BC00472=140020,825224,1075175
BC00473=143607,831260,1075175
BC00474=145042,833675,1075175
BC00475=145042,833669,1075175
BC00476=143607,831255,1075175
BC00477=140021,825218,1075175
BC00478=140020,825224,1075175
BC00479=325300,955877,1075175
BC00480=326098,960603,1075175
BC00481=326417,962494,1075175
BC00482=373942,970744,1075175
BC00483=373623,968854,1075175
BC00484=372825,964128,1075175
BC00485=388713,844195,1075175
BC00486=388713,844195,1075175
BC00487=388713,844195,1075175
BC00488=388713,844195,1075175
BC00489=388713,844195,1075175
BC00490=392621,845560,1075175
BC00491=388844,869736,1075175
BC00492=388844,869736,1075175
BC00493=388844,869736,1075175
BC00494=388844,869736,1075175
BC00495=386515,859937,1075175
BC00496=382579,861240,1075175
BC00497=382579,861240,1075175
BC00498=398174,862085,1075175
BC00499=398174,860729,1075175
BC00500=398175,860364,1075172
BC00501=398174,860364,1075175
BC00502=398174,860364,1075175
BC00503=398174,860364,1075175
BC00504=398174,859798,1075175
BC00505=398174,853900,1075175
BC00506=335556,962122,1075175
BC00507=313093,960913,1075175
BC00508=312779,966350,1075175
BC00509=312653,968525,1075175
BC00510=317356,969341,1075175
BC00511=322596,970251,1075175
BC00512=322722,968076,1075175
BC00513=323035,962639,1075175
BC00514=275790,965253,1075175
BC00515=219096,968390,1075175
BC00516=223120,970377,1075175
BC00517=224729,971172,1075175
BC00518=220819,966503,1075175
BC00519=219210,965708,1075175
BC00520=215186,963721,1075175
BC00521=283252,975030,1075175
BC00522=343583,985054,1075175
BC00523=351318,986339,1075175
BC00524=346951,987672,1075175
BC00525=345577,987893,1075175
BC00526=346840,986833,1075175
BC00527=348087,985787,1075175
BC00528=349722,984415,1075175
BC00529=349722,984415,1075175
BC00530=349722,984415,1075175
BC00531=351469,983882,1075175
BC00532=355836,982549,1075175
BC00533=351318,986339,1075175
BC00534=322594,894090,1075175
BC00535=319270,885244,1075175
BC00536=319145,881395,1075175
BC00537=319096,879856,1075175
BC00538=319096,879856,1075175
BC00539=310158,881364,1075175
BC00540=310282,885213,1075175
BC00541=287932,898047,1075175
BC00542=289217,893542,1075175
BC00543=289730,891739,1075175
BC00544=285692,891718,1075175
BC00545=285179,893520,1075175
BC00546=283894,898026,1075175
BC00547=317886,904348,1075175
BC00548=321408,904356,1075175
BC00549=251917,914686,1075175
BC00550=191223,885215,1075175
BC00551=191223,923708,1075175
BC00552=186619,926680,1075175
BC00553=184777,927869,1075175
BC00554=132357,904545,1075175
BC00555=148459,907340,1075175
BC00556=150318,907039,1075175
BC00557=172119,903510,1075175
BC00558=172334,901853,1075175
BC00559=172871,897709,1075175
BC00560=285135,920733,1075175
BC00561=282294,924718,1075175
BC00562=278369,925274,1075175
BC00563=250842,915028,1075175
BC00564=302481,924098,1075175
BC00565=235391,926007,1075175
BC00566=233206,924435,1075175
BC00567=227742,920504,1075175
BC00568=172871,874776,1075175
BC00569=140749,823212,1075175
BC00570=114392,780903,1075175
BC00571=114392,780903,1075175
BC00572=114392,780903,1075175
BC00573=114392,780903,1075175
BC00574=114392,780903,1075175
BC00575=114392,780903,1075175
BC00576=114392,780903,1075175
BC00577=114392,780903,1075175
BC00578=147421,791636,1075175
BC00579=157474,794903,1075175
BC00580=157474,794903,1075175
BC00581=157474,794903,1075175
BC00582=157474,794903,1075175
BC00583=157474,794903,1075175
BC00584=157474,794903,1075175
BC00585=157474,794903,1075175
BC00586=157474,794903,1075175
BC00587=188976,808930,1075175
BC00588=188976,808930,1075175
BC00589=188976,808930,1075175
BC00590=188976,808930,1075175
BC00591=188976,808930,1075175
BC00592=188976,808930,1075175
BC00593=188976,808930,1075175
BC00594=188976,808930,1075175
BC00595=147641,782026,1075175
BC00596=198576,845167,1075175
BC00597=232811,933878,1075175
BC00598=232896,933343,1075175
BC00599=232035,938717,1075175
BC00600=231691,940867,1075175
BC00601=233684,941999,1075172
BC00602=218918,951560,1075175
BC00603=218487,945823,1075175
BC00604=199715,965567,1075175
BC00605=202231,971242,1075175
BC00606=203237,973512,1075175
BC00607=199770,971953,1075175
BC00608=198686,969649,1075175
BC00609=195975,963887,1075175
BC00610=268319,958805,1075175
BC00611=299772,956595,1075175
BC00612=294961,960779,1075175
BC00613=302025,967105,1075175
BC00614=302025,967105,1075175
BC00615=302862,967571,1075175
BC00616=304981,965989,1075175
BC00617=310277,962032,1075175
BC00618=299772,946803,1075175
BC00619=156368,867370,1075175
BC00620=114190,943890,1075175
BC00621=112857,947238,1075175
BC00622=112324,948578,1075175
BC00623=57438,939049,1075175
BC00624=57438,939049,1075175
BC00625=57972,937710,1075175
BC00626=59304,934362,1075175
BC00627=59959,931573,1075175
BC00628=60163,930702,1075175
BC00629=64900,934429,1075175
BC00630=66794,935919,1075175
BC00631=70926,933782,1075175
BC00632=86714,920781,1075175
BC00633=88876,916896,1075175
BC00634=87247,915034,1075175
BC00635=83174,910378,1075175
BC00636=93083,910762,1075175
BC00637=96362,916987,1075175
BC00638=97673,919477,1075175
BC00639=102107,915596,1075175
BC00640=93734,925368,1075175
BC00641=92128,923198,1075175
BC00642=88115,917772,1075175
BC00643=59304,853852,1075175
BC00644=302197,956351,1075175
BC00645=302197,956351,1075175
BC00646=297684,958955,1075175
BC00647=295879,959997,1075175
BC00648=304739,998959,1075175
BC00649=304723,978619,1075175
BC00650=293949,1042099,1075175
BC00651=295296,1044279,1075175
BC00652=298665,1049727,1075175
BC00653=298665,1049727,1075175
BC00654=21214,672831,1075175
BC00655=78393,670967,1075175
BC00656=177059,727519,1002542
BC00657=78393,913126,1075175
BC00658=70793,903989,1075175
BC00659=70793,903989,1075175
BC00660=70793,903989,1075175
BC00661=70793,903989,1075175
BC00662=70793,903989,1075175
BC00663=70793,903989,1075175
BC00664=70793,903989,1075175
BC00665=70793,903989,1075175
BC00666=70793,903989,1075175
BC00667=103901,897249,1075175
BC00668=103901,897249,1075175
BC00669=103901,897249,1075175
BC00670=103901,897249,1075175
BC00671=103901,897249,1075175
BC00672=103901,897249,1075175
BC00673=103901,897249,1075175
BC00674=103901,897249,1075175
BC00675=89915,910531,1075175
BC00676=89915,910531,1075175
BC00677=89916,910530,1075174
BC00678=89916,910530,1075174
BC00679=89916,910530,1075174
BC00680=89916,910530,1075174
BC00681=89916,910530,1075174
BC00682=89916,910530,1075174
BC00683=89916,910530,1075174
BC00684=89915,910531,1075175
BC00685=89915,910531,1075175
BC00686=89915,910531,1075175
BC00687=89915,910531,1075175
BC00688=89915,910531,1075175
BC00689=89915,910531,1075175
BC00690=89915,910531,1075175
BC00691=27368,899646,1075175
BC00692=27368,899646,1075175
BC00693=27368,899646,1075175
BC00694=27368,899646,1075175
BC00695=27368,899646,1075175
BC00696=27368,899646,1075175
BC00697=27368,899646,1075175
BC00698=27368,899646,1075175
BC00699=160753,772187,1075175
BC00700=160753,772187,1075175
BC00701=160753,772187,1075175
BC00702=160753,772187,1075175
BC00703=160753,772187,1075175
BC00704=160753,772187,1075175
BC00705=160753,772187,1075175
BC00706=160753,772187,1075175
BC00707=160753,772187,1075175
BC00708=160753,772187,1075175
BC00709=160753,772187,1075175
BC00710=160753,772187,1075175
BC00711=123402,765716,1075175
BC00712=123402,765716,1075175
BC00713=123402,765716,1075175
BC00714=123402,765716,1075175
BC00715=123402,765716,1075175
BC00716=123402,765716,1075175
BC00717=123402,765716,1075175
BC00718=123402,765716,1075175
BC00719=123402,765716,1075175
BC00720=123402,765716,1075175
BC00721=123402,765716,1075175
BC00722=129464,768278,1075175
BC00723=151149,777443,1075175
BC00724=169689,785624,1075175
BC00725=169689,785624,1075175
BC00726=169689,785624,1075175
BC00727=169689,785624,1075175
BC00728=169689,785624,1075175
BC00729=169689,785624,1075175
BC00730=169689,785624,1075175
BC00731=169689,785624,1075175
BC00732=169689,785624,1075175
BC00733=169689,785624,1075175
BC00734=169689,785624,1075175
BC00735=169689,785624,1075175
BC00736=169689,785624,1075175
BC00737=120114,813651,1075175
BC00738=120114,813651,1075175
BC00739=120114,813651,1075175
BC00740=120114,813651,1075175
BC00741=120114,813651,1075175
BC00742=120114,813651,1075175
BC00743=120114,813651,1075175
BC00744=120114,813651,1075175
BC00745=120114,813651,1075175
BC00746=120114,813651,1075175
BC00747=120114,813651,1075175
BC00748=120114,813651,1075175
BC00749=120114,813651,1075175
BC00750=141881,838168,1075175
BC00751=141881,838168,1075175
BC00752=141881,838168,1075175
BC00753=141881,838168,1075175
BC00754=141881,838168,1075175
BC00755=141881,838168,1075175
BC00756=141881,838168,1075175
BC00757=141881,838168,1075175
BC00758=141881,838168,1075175
BC00759=141881,838168,1075175
BC00760=141881,838168,1075175
BC00761=141881,838168,1075175
BC00762=141881,838168,1075175
BC00763=69874,805894,1075175
BC00764=70019,750208,1075175
BC00765=70019,750208,1075175
BC00766=70019,750208,1075175
BC00767=70019,750208,1075175
BC00768=70019,750208,1075175
BC00769=70019,750208,1075175
BC00770=70019,750208,1075175
BC00771=70019,750208,1075175
BC00772=70019,750208,1075175
BC00773=70019,750208,1075175
BC00774=70019,750208,1075175
BC00775=70019,750208,1075175
BC00776=70019,750208,1075175
BC00777=70018,750208,1075172
BC00778=70018,750208,1075172
BC00779=70018,750208,1075172
BC00780=70018,750208,1075172
BC00781=70018,750208,1075172
BC00782=70018,750208,1075172
BC00783=70018,750208,1075172
BC00784=70018,750208,1075172
BC00785=110204,822960,1075174
BC00786=128430,855958,1075175
BC00787=125005,945340,1075175
BC00788=125005,945340,1075175
BC00789=125005,945340,1075175
BC00790=125005,945340,1075175
BC00791=125005,945340,1075175
BC00792=125005,945340,1075175
BC00793=125005,945340,1075175
BC00794=125005,945340,1075175
BC00795=125005,945340,1075175
BC00796=125005,945340,1075175
BC00797=125005,945340,1075175
BC00798=177748,940008,1075175
BC00799=177748,940008,1075175
BC00800=177748,940008,1075175
BC00801=177748,940008,1075175
BC00802=177748,940008,1075175
BC00803=177748,940008,1075175
BC00804=177748,940008,1075175
BC00805=177748,940008,1075175
BC00806=177748,940008,1075175
BC00807=177748,940008,1075175
BC00808=177748,940008,1075175
BC00809=177748,940008,1075175
BC00810=225975,953000,1075175
BC00811=225975,953000,1075175
BC00812=225975,953000,1075175
BC00813=225975,953000,1075175
BC00814=225975,953000,1075175
BC00815=225975,953000,1075175
BC00816=225975,953000,1075175
BC00817=225975,953000,1075175
BC00818=225975,953000,1075175
BC00819=225975,953000,1075175
BC00820=225975,953000,1075175
BC00821=225975,953000,1075175
BC00822=254413,953027,1075175
BC00823=252547,954523,1075175
BC00824=252548,954519,1075175
BC00825=252583,954651,1075175
BC00826=252019,957675,1075175
BC00827=252583,954651,1075175
BC00828=252165,954787,1075175
BC00829=249030,954243,1075175
BC00830=252165,954787,1075175
BC00831=258696,949550,1075175
BC00832=257059,950024,1075175
BC00833=265795,953000,1075175
BC00834=265795,953000,1075175
BC00835=265795,953000,1075175
BC00836=265795,953000,1075175
BC00837=265795,953000,1075175
BC00838=265795,953000,1075175
BC00839=265795,953000,1075175
BC00840=265795,953000,1075175
BC00841=265795,953000,1075175
BC00842=265795,953000,1075175
BC00843=265795,953000,1075175
BC00844=254634,951648,1075175
BC00845=253737,956448,1075175
BC00846=253378,958368,1075175
BC00847=253379,958364,1075175
BC00848=253259,958395,1075175
BC00849=252695,961419,1075175
BC00850=253259,958395,1075175
BC00851=254515,951675,1075175
BC00852=248439,993035,1075175
BC00853=271638,1017285,1075175
BC00854=314947,1062557,1075175
BC00855=311280,1056373,1075175
BC00856=310409,1054905,1075175
BC00857=310409,1054901,1075175
BC00858=310409,1054905,1075175
BC00859=284329,1066137,1075175
BC00860=285931,1063482,1075175
BC00861=284329,1066137,1075175
BC00862=333588,1039325,1075175
BC00863=330835,1037779,1075175
BC00864=333588,1039325,1075175
BC00865=340460,1045393,1075175
BC00866=319968,1046454,1075175
BC00867=279319,1048558,1075175
BC00868=281895,1044284,1075175
BC00869=282926,1042574,1075175
BC00870=282926,1042570,1075175
BC00871=282744,1042486,1075175
BC00872=284346,1039831,1075175
BC00873=282744,1042486,1075175
BC00874=279137,1048470,1075175
BC00875=253507,1028204,1074244
BC00876=253507,1028204,1074244
BC00877=253507,1028204,1074244
BC00878=253507,1028204,1074244
BC00879=253507,1028204,1074244
BC00880=253507,1028204,1074244
BC00881=253507,1028204,1074244
BC00882=253507,1028204,1074244
BC00883=253507,1028204,1074244
BC00884=253507,1028204,1074244
BC00885=253507,1028204,1074244
BC00886=253507,1028204,1074244
BC00887=253507,1028204,1074244
BC00888=212842,1022781,1075175
BC00889=146334,1015862,1075175
BC00890=66205,1045023,1075175
BC00891=66205,1045023,1075175
BC00892=66205,1045023,1075175
BC00893=66205,1045023,1075175
BC00894=66205,1045023,1075175
BC00895=66205,1045023,1075175
BC00896=66205,1045023,1075175
BC00897=66205,1045023,1075175
BC00898=66205,1045023,1075175
BC00899=66205,1045023,1075175
BC00900=66205,1045023,1075175
BC00901=66205,1045023,1075175
BC00902=125029,959783,1075175
BC00903=190390,972133,1075175
BC00904=190390,972133,1075175
BC00905=190390,972133,1075173
BC00906=190390,972133,1075175
BC00907=190390,972133,1075175
BC00908=190390,972133,1075175
BC00909=190390,972133,1075175
BC00910=190390,972133,1075175
BC00911=190390,972133,1075175
BC00912=190390,972133,1075175
BC00913=190390,972133,1075175
BC00914=190390,972133,1075175
BC00915=190390,972133,1075175
BC00916=103363,888035,1075175
BC00917=35304,822265,1075175
BC00918=35304,822265,1075175
BC00919=35304,822265,1075175
BC00920=35304,822265,1075175
BC00921=35304,822265,1075175
BC00922=35304,822265,1075175
BC00923=35304,822265,1075175
BC00924=35304,822265,1075175
BC00925=35304,822265,1075175
BC00926=35304,822265,1075175
BC00927=35304,822265,1075175
BC00928=35304,822265,1075175
BC00929=167967,799945,1075175
BC00930=311305,898961,1075175
BC00931=311305,898961,1075175
BC00932=311305,898961,1075175
BC00933=311305,898961,1075175
BC00934=311305,898961,1075175
BC00935=311305,898961,1075175
BC00936=311305,898961,1075175
BC00937=311305,898961,1075175
BC00938=311305,898961,1075175
BC00939=311305,898961,1075175
BC00940=311305,898961,1075175
BC00941=311305,898961,1075175
BC00942=113180,824290,1075229
BC00943=113180,824290,1075229
BC00944=113180,824290,1075229
BC00945=113180,824290,1075229
BC00946=113180,824290,1075229
BC00947=113180,824290,1075229
BC00948=113180,824290,1075229
BC00949=113180,824290,1075229
BC00950=113180,824290,1075229
BC00951=113180,824290,1075229
BC00952=113180,824290,1075229
BC00953=113180,824290,1075229
BC00954=355762,967535,1075175
BC00955=355762,967535,1075175
BC00956=355762,967535,1075175
BC00957=355762,967535,1075175
BC00958=355762,967535,1075175
BC00959=355762,967535,1075175
BC00960=355762,967535,1075175
BC00961=355762,967535,1075175
BC00962=397203,974799,1075175
BC00963=397203,974799,1075175
BC00964=397203,974799,1075175
BC00965=397203,974799,1075175
BC00966=397203,974799,1075175
BC00967=397203,974799,1075175
BC00968=397203,974799,1075175
BC00969=397203,974799,1075175
BC00970=389868,1004990,1075175
BC00971=389868,1004990,1075175
BC00972=389868,1004990,1075175
BC00973=389868,1004990,1075175
BC00974=389868,1004990,1075175
BC00975=389868,1004990,1075175
BC00976=397203,974799,1075175
BC00977=279782,952911,1075175
BC00978=264332,967435,1075175
BC00979=264332,967435,1075175
BC00980=264332,967435,1075175
BC00981=264332,967435,1075175
BC00982=264332,967435,1075175
BC00983=264332,967435,1075175
BC00984=264332,967435,1075175
BC00985=264332,967435,1075175
BC00986=264332,967435,1075175
BC00987=264332,967435,1075175
BC00988=264332,967435,1075175
BC00989=290594,956201,1075175
BC00990=316856,944967,1075175
BC00991=316856,944967,1075175
BC00992=316856,944967,1075175
BC00993=316856,944967,1075175
BC00994=316856,944967,1075175
BC00995=316856,944967,1075175
BC00996=316856,944967,1075175
BC00997=316856,944967,1075175
BC00998=316856,944967,1075175
BC00999=316856,944967,1075175
BC01000=316856,944967,1075175
BC01001=316856,944967,1075175
BC01002=316856,944967,1075175
BC01003=316856,944967,1075175
BC01004=316856,944967,1075175
BC01005=316856,944967,1075175
BC01006=329946,891084,1075175
BC01007=337525,859888,1075175
BC01008=337525,859888,1075175
BC01009=337525,859888,1075175
BC01010=337525,859888,1075175
BC01011=337525,859888,1075175
BC01012=337525,859888,1075175
BC01013=337525,859888,1075175
BC01014=337525,859888,1075175
BC01015=238148,874377,1075175
BC01016=227206,875826,1075175
BC01017=227206,875826,1075175
BC01018=227206,875826,1075175
BC01019=227206,875826,1075175
BC01020=227206,875826,1075175
BC01021=227206,875826,1075175
BC01022=280946,887675,1075175
BC01023=280946,887675,1075175
BC01024=280946,887675,1075175
BC01025=280946,887675,1075175
BC01026=280946,887675,1075175
BC01027=280946,887675,1075175
BC01028=280946,887675,1075175
BC01029=280946,887675,1075175
BC01030=239261,850045,1075175
BC01031=207869,857354,1075175
BC01032=207869,857354,1075175
BC01033=207869,857354,1075175
BC01034=207869,857354,1075175
BC01035=207869,857354,1075175
BC01036=207869,857354,1075175
BC01037=207869,857354,1075175
BC01038=207869,857354,1075175
BC01039=207996,857850,1075175
BC01040=184532,936508,1075175
BC01041=203495,1021788,1075175
BC01042=203934,1024782,1075175
BC01043=204108,1022909,1075171
BC01044=204109,1022908,1075172
BC01045=193998,1019034,1075175
BC01046=193559,1023720,1075175
BC01047=122539,997675,1075175
BC01048=122539,997675,1075175
BC01049=122540,997675,1075169
BC01050=122540,997675,1075169
BC01051=122539,997675,1075175
BC01052=122539,997675,1075175
BC01053=110261,971952,1075175
BC01054=110261,971952,1075175
BC01055=110261,971952,1075175
BC01056=110261,971952,1075175
BC01057=110261,971952,1075175
BC01058=110261,971952,1075175
BC01059=222038,980891,1075175
BC01060=314817,1023461,1075175
BC01061=333143,1031869,1075175
BC01062=333143,1031869,1075175
BC01063=333143,1031869,1075175
BC01064=333143,1031869,1075175
BC01065=333143,1031869,1075175
BC01066=163675,1006427,1075175
BC01067=163675,1006427,1075175
BC01068=164114,1001741,1075175
BC01069=164289,999867,1075175
BC01070=160191,997498,1075175
BC01071=158450,996490,1075175
BC01072=154353,994119,1075175
BC01073=154178,995993,1075175
BC01074=153739,1000679,1075175
BC01075=82719,974634,1075175
BC01076=82719,974634,1075175
BC01077=82720,974634,1075172
BC01078=82720,974634,1075172
BC01079=82719,974634,1075175
BC01080=82720,974634,1075173
BC01081=82719,974634,1075175
BC01082=82719,974634,1075175
BC01083=70441,948911,1075175
BC01084=70441,948911,1075175
BC01085=70441,948911,1075175
BC01086=70441,948911,1075175
BC01087=70441,948911,1075175
BC01088=70441,948911,1075175
BC01089=182218,957850,1075175
BC01090=274997,1000420,1075175
BC01091=293323,1008828,1075175
BC01092=293323,1008828,1075175
BC01093=293323,1008828,1075175
BC01094=293323,1008828,1075175
BC01095=293323,1008828,1075175
BC01096=293323,1008828,1075175
BC01097=337244,1059629,1075175
BC01098=337244,1059629,1075175
BC01099=337244,1059629,1075175
BC01100=337244,1059629,1075175
BC01101=337244,1059629,1075175
BC01102=337244,1059629,1075175
BC01103=337244,1059629,1075175
BC01104=227430,982125,1075175
BC01105=115014,939685,1075175
BC01106=118867,937244,1075175
BC01107=120408,936268,1075175
BC01108=140995,947826,1075175
BC01109=182041,976368,1075175
BC01110=180846,977671,1075175
BC01111=177859,980929,1075175
BC01112=194800,984537,1075175
BC01113=244653,1016084,1075175
BC01114=241511,1010564,1075175
BC01115=240254,1008357,1075175
BC01116=240254,1008354,1075175
BC01117=241511,1010562,1075175
BC01118=244653,1016081,1075175
BC01119=244653,1016084,1075175
BC01120=272695,1033702,1075175
BC01121=285514,1041756,1075175
BC01122=284751,1045931,1075175
BC01123=282162,1039999,1075175
BC01124=281126,1037626,1075175
BC01125=207140,1028015,1075175
BC01126=213441,1031536,1075175
BC01127=213388,1030834,1075175
BC01128=213388,1030834,1075175
BC01129=212628,1031081,1075217
BC01130=212628,1031081,1075217
BC01131=212628,1031081,1075217
BC01132=212628,1031081,1075217
BC01133=212628,1031081,1075202
BC01134=202210,1012854,1075175
BC01135=202210,1012854,1075175
BC01136=196613,982513,1075175
BC01137=175963,870568,1075175
BC01138=163612,803610,1075175
BC01139=152631,778532,1075175
BC01140=146092,780306,1075175
BC01141=143477,781016,1075175
BC01142=143597,781078,1075175
BC01143=143625,781092,1075175
BC01144=143746,781156,1075175
BC01145=146361,780446,1075175
BC01146=152900,778672,1075175
BC01147=152900,778672,1075175
BC01148=74084,744686,1075175
BC01149=74084,744686,1075175
BC01150=67287,679894,1075175
BC01151=67287,679894,1075175
BC01152=67287,679894,1075175
BC01153=67287,679894,1075175
BC01154=67287,679894,1075175
BC01155=67287,679894,1075175
BC01156=67287,679894,1075175
BC01157=67287,679894,1075175
BC01158=83395,694294,1075175
BC01159=102108,711022,1075175
BC01160=165558,767742,1075175
BC01161=222482,818628,1075175
BC01162=215814,820321,1075175
BC01163=213147,820999,1075175
BC01164=213147,820994,1075175
BC01165=213147,820993,1075175
BC01166=213148,820988,1075175
BC01167=215815,820311,1075175
BC01168=222483,818617,1075175
BC01169=173722,816110,1075175
BC01170=90356,811823,1075175
BC01171=89696,811574,1075175
BC01172=89432,811475,1075175
BC01173=89432,811475,1075175
BC01174=89432,811475,1075175
BC01175=85301,809160,1075175
BC01176=73323,802435,1075175
BC01177=69196,800114,1075175
BC01178=69460,800213,1075175
BC01179=70120,800462,1075175
BC01180=203969,867991,1075175
BC01181=200192,866637,1075175
BC01182=198681,866095,1075175
BC01183=196278,870078,1075175
BC01184=188025,883752,1075175
BC01185=185620,887734,1075175
BC01186=187131,888276,1075175
BC01187=190907,889630,1075175
BC01188=185807,834457,1075175
BC01189=185042,826181,1075175
BC01190=182820,831186,1075175
BC01191=181931,833188,1075175
BC01192=205283,846231,1075175
BC01193=246906,863634,1075175
BC01194=246906,863634,1075175
BC01195=248214,861732,1075175
BC01196=251484,856977,1075175
BC01197=177002,833071,1075175
BC01198=153563,828435,1075175
BC01199=140020,825224,1075175
BC01200=143607,831260,1075175
BC01201=145042,833675,1075175
BC01202=145042,833669,1075175
BC01203=143607,831255,1075175
BC01204=140021,825218,1075175
BC01205=140020,825224,1075175
BC01206=325300,955877,1075175
BC01207=326098,960603,1075175
BC01208=326417,962494,1075175
BC01209=373942,970744,1075175
BC01210=373934,970699,1075175
BC01211=373927,970659,1075175
BC01212=372825,964128,1075175
BC01213=388713,844195,1075175
BC01214=388713,844195,1075175
BC01215=388713,844195,1075175
BC01216=388713,844195,1075175
BC01217=388713,844195,1075175
BC01218=392621,845560,1075175
BC01219=388844,869736,1075175
BC01220=388844,869736,1075175
BC01221=388844,869736,1075175
BC01222=388844,869736,1075175
BC01223=386515,859937,1075175
BC01224=382579,861240,1075175
BC01225=382579,861240,1075175
BC01226=398174,862085,1075175
BC01227=398174,860729,1075175
BC01228=398175,860364,1075172
BC01229=398174,860364,1075175
BC01230=398174,860364,1075175
BC01231=398174,860364,1075175
BC01232=398174,859798,1075175
BC01233=398174,853900,1075175
BC01234=335556,962122,1075175
BC01235=313093,960913,1075175
BC01236=312779,966350,1075175
BC01237=312653,968525,1075175
BC01238=317356,969341,1075175
BC01239=322596,970251,1075175
BC01240=322722,968076,1075175
BC01241=323035,962639,1075175
BC01242=275790,965253,1075175
BC01243=219096,968390,1075175
BC01244=223120,970377,1075175
BC01245=224729,971172,1075175
BC01246=220819,966503,1075175
BC01247=219210,965708,1075175
BC01248=215186,963721,1075175
BC01249=283252,975030,1075175
BC01250=343583,985054,1075175
BC01251=351318,986339,1075175
BC01252=346951,987672,1075175
BC01253=345577,987893,1075175
BC01254=346840,986833,1075175
BC01255=348087,985787,1075175
BC01256=349722,984415,1075175
BC01257=349722,984415,1075175
BC01258=349722,984415,1075175
BC01259=351469,983882,1075175
BC01260=355836,982549,1075175
BC01261=351318,986339,1075175
BC01262=375376,962122,1075175
BC01263=352913,960913,1075175
BC01264=352599,966350,1075175
BC01265=352473,968525,1075175
BC01266=357176,969341,1075175
BC01267=362416,970251,1075175
BC01268=362542,968076,1075175
BC01269=362855,962639,1075175
BC01270=315610,965253,1075175
BC01271=258916,968390,1075175
BC01272=262940,970377,1075175
BC01273=264549,971172,1075175
BC01274=260639,966503,1075175
BC01275=259030,965708,1075175
BC01276=255006,963721,1075175
BC01277=323072,975030,1075175
BC01278=383403,985054,1075175
BC01279=391138,986339,1075175
BC01280=386771,987672,1075175
BC01281=385397,987893,1075175
BC01282=386660,986833,1075175
BC01283=387907,985787,1075175
BC01284=389542,984415,1075175
BC01285=389542,984415,1075175
BC01286=389542,984415,1075175
BC01287=391289,983882,1075175
BC01288=394785,983280,1075175
BC01289=393350,984484,1075175
BC01290=322594,894090,1075175
BC01291=319270,885244,1075175
BC01292=319145,881395,1075175
BC01293=319096,879856,1075175
BC01294=319096,879856,1075175
BC01295=310158,881364,1075175
BC01296=310282,885213,1075175
BC01297=287932,898047,1075175
BC01298=289217,893542,1075175
BC01299=289730,891739,1075175
BC01300=285692,891718,1075175
BC01301=285179,893520,1075175
BC01302=283894,898026,1075175
BC01303=317886,904348,1075175
BC01304=321408,904356,1075175
BC01305=251917,914686,1075175
BC01306=191223,885215,1075175
BC01307=191223,923708,1075175
BC01308=186619,926680,1075175
BC01309=184777,927869,1075175
BC01310=132357,904545,1075175
BC01311=148459,907340,1075175
BC01312=150318,907039,1075175
BC01313=172119,903510,1075175
BC01314=172334,901853,1075175
BC01315=172871,897709,1075175
BC01316=285135,920733,1075175
BC01317=282294,924718,1075175
BC01318=278369,925274,1075175
BC01319=250842,915028,1075175
BC01320=259644,916574,1075175
BC01321=259644,916574,1075174
BC01322=259644,916574,1075175
BC01323=285135,920733,1075175
BC01324=320470,920733,1075175
BC01325=320470,920733,1075175
BC01326=320470,920733,1075172
BC01327=320470,920733,1075172
BC01328=320470,920733,1075172
BC01329=302481,924098,1075175
BC01330=235391,926007,1075175
BC01331=235391,926007,1075175
BC01332=227742,920504,1075175
BC01333=172871,874776,1075175
BC01334=140749,823212,1075175
BC01335=114392,780903,1075175
BC01336=114392,780903,1075175
BC01337=114392,780903,1075175
BC01338=114392,780903,1075175
BC01339=114392,780903,1075175
BC01340=114392,780903,1075175
BC01341=114392,780903,1075175
BC01342=114392,780903,1075175
BC01343=147421,791636,1075175
BC01344=157474,794903,1075175
BC01345=157474,794903,1075175
BC01346=157474,794903,1075175
BC01347=157474,794903,1075175
BC01348=157474,794903,1075175
BC01349=157474,794903,1075175
BC01350=157474,794903,1075175
BC01351=157474,794903,1075175
BC01352=188976,808930,1075175
BC01353=188976,808930,1075175
BC01354=188976,808930,1075175
BC01355=188976,808930,1075175
BC01356=188976,808930,1075175
BC01357=188976,808930,1075175
BC01358=188976,808930,1075175
BC01359=188976,808930,1075175
BC01360=147641,782026,1075175
BC01361=198576,845167,1075175
BC01362=232811,933878,1075175
BC01363=232896,933343,1075175
BC01364=232035,938717,1075175
BC01365=231691,940867,1075175
BC01366=233684,941999,1075172
BC01367=218918,951560,1075175
BC01368=218487,945823,1075175
BC01369=199715,965567,1075175
BC01370=202231,971242,1075175
BC01371=203237,973512,1075175
BC01372=199770,971953,1075175
BC01373=198686,969649,1075175
BC01374=195975,963887,1075175
BC01375=268319,958805,1075175
BC01376=299772,956595,1075175
BC01377=294961,960779,1075175
BC01378=302025,967105,1075175
BC01379=302025,967105,1075175
BC01380=302862,967571,1075175
BC01381=304981,965989,1075175
BC01382=310277,962032,1075175
BC01383=299772,946803,1075175
BC01384=156368,867370,1075175
BC01385=114190,943890,1075175
BC01386=112857,947238,1075175
BC01387=112324,948578,1075175
BC01388=112324,948578,1075175
BC01389=91893,945031,1075175
BC01390=58795,939285,1075175
BC01391=57438,939049,1075175
BC01392=57972,937710,1075175
BC01393=59304,934362,1075175
BC01394=59959,931573,1075175
BC01395=60163,930702,1075175
BC01396=64900,934429,1075175
BC01397=66794,935919,1075175
BC01398=70926,933782,1075175
BC01399=86714,920781,1075175
BC01400=88876,916896,1075175
BC01401=87247,915034,1075175
BC01402=83174,910378,1075175
BC01403=93083,910762,1075175
BC01404=96362,916987,1075175
BC01405=97673,919477,1075175
BC01406=102107,915596,1075175
BC01407=93734,925368,1075175
BC01408=92128,923198,1075175
BC01409=88115,917772,1075175
BC01410=59304,853852,1075175
BC01411=302197,956351,1075175
BC01412=302197,956351,1075175
BC01413=297684,958955,1075175
BC01414=295879,959997,1075175
BC01415=304739,998959,1075175
BC01416=304723,978619,1075175
BC01417=293949,1042099,1075175
BC01418=295296,1044279,1075175
BC01419=298665,1049727,1075175
BC01420=298665,1049727,1075175
BC01421=302197,956351,1075175
BC01422=339931,956351,1075175
BC01423=339931,956351,1075175
BC01424=339931,956351,1075175
BC01425=345108,996833,1075175
BC01426=329498,1037164,1075167
BC01427=329498,1037164,1075167
BC01428=329498,1037164,1075167
BC01429=326051,1024211,1075168
BC01430=315665,949153,1075168
BC01431=252444,896504,1075168
BC01432=116643,896504,1075168
BC01433=116643,972299,1075168
BC01434=116644,972299,1070754
BC01435=116644,972299,1070754
BC01436=121804,1001122,1070754
BC01437=121804,1001122,1070754
BC01438=121804,1001122,1070754
BC01439=121804,1001122,1070754
BC01440=164206,909682,1070754
BC01441=118737,834368,1072160
BC01442=21214,672831,1075175
BC01443=21214,672831,272422
BC01444=236199,677421,175874
BC01445=277013,737492,108841
BC01446=313151,790681,49489
BC01447=313151,790681,49489
BC01448=313151,790681,49489
BC01449=313151,790681,49489
BC01450=313151,790681,49489
BC01451=313151,790681,49489
BC01452=313151,790681,49489
BC01453=313151,790681,49489
BC01454=313151,790681,49489
BC01455=313151,790681,49489
BC01456=313151,790681,49489
BC01457=313151,790681,49489
BC01458=313151,790681,49489
BC01459=339082,790681,219047
BC01460=339082,790681,219047
BC01461=339082,790681,219047
BC01462=339082,790681,219047
BC01463=339082,790681,219047
BC01464=339082,790681,219047
BC01465=339082,790681,219047
BC01466=339082,790681,219047
BC01467=339082,790681,219047
BC01468=318756,790681,206942
BC01469=318756,790681,206942
BC01470=318756,790681,206942
BC01471=318756,790681,206942
BC01472=318756,790681,206942
BC01473=318756,790681,206942
BC01474=318756,790681,206941
BC01475=318756,790681,206941
BC01476=318756,790681,206942
BC01477=330178,790681,186109
BC01478=360333,790681,131110
BC01479=360333,790681,131110
BC01480=360333,790681,131110
BC01481=360333,790681,131110
BC01482=360333,790681,131110
BC01483=360333,790681,131110
BC01484=360333,790681,131110
BC01485=360333,790681,131110
BC01486=360333,790681,131110
BC01487=319787,790681,204440
BC01488=319787,790681,204440
BC01489=319787,790681,204440
BC01490=319787,790681,204440
BC01491=319787,790681,204440
BC01492=319787,790681,204440
BC01493=319787,790681,204440
BC01494=319787,790681,204440
BC01495=319787,790681,204440
BC01496=319787,790681,204440
BC01497=319787,790681,204440
BC01498=319787,790681,204440
BC01499=319787,790681,204440
BC01500=319787,790681,204440
BC01501=319787,790681,204440
BC01502=319787,790681,204440
BC01503=345989,790681,139065
BC01504=345989,790681,139065
BC01505=345988,790681,139065
BC01506=345988,790681,139065
BC01507=345988,790681,139065
BC01508=345988,790681,139065
BC01509=345988,790681,139065
BC01510=345988,790681,139065
BC01511=345988,790681,139065
BC01512=345988,790681,139065
BC01513=345988,790681,139065
BC01514=345988,790681,139065
BC01515=345988,790681,139065
BC01516=345988,790681,139065
BC01517=345988,790681,139065
BC01518=345989,790681,139065
BC01519=308625,748445,196549
BC01520=237635,668196,305769
BC01521=196160,672502,403752
BC01522=196160,672502,403752
BC01523=196160,727236,321537
BC01524=196160,765129,264619
BC01525=196160,765129,264619
BC01526=196160,765129,264619
BC01527=196160,765129,264619
BC01528=196160,765129,264619
BC01529=196160,765129,264619
BC01530=196160,765129,264619
BC01531=196160,765129,264619
BC01532=196160,765129,264619
BC01533=196160,765129,264619
BC01534=196160,765129,264619
BC01535=196160,765129,264619
BC01536=196160,765129,264619
BC01537=196160,765129,264619
BC01538=196160,765129,264619
BC01539=196160,765129,264619
BC01540=172117,778418,210988
BC01541=172117,778418,210988
BC01542=172117,778418,210988
BC01543=172117,778418,210988
BC01544=172117,778418,210988
BC01545=172117,778418,210988
BC01546=172117,778418,210988
BC01547=172117,778418,210988
BC01548=172117,778418,210988
BC01549=172117,778418,210988
BC01550=172117,778418,210988
BC01551=172117,778418,210988
BC01552=172117,778418,210988
BC01553=172117,778418,210988
BC01554=172117,778418,210988
BC01555=172117,778418,210988
BC01556=149065,790681,133702
BC01557=149065,790681,133702
BC01558=149065,790681,133702
BC01559=149065,790681,133702
BC01560=149065,790681,133702
BC01561=149065,790681,133702
BC01562=149065,790681,133702
BC01563=149065,790681,133702
BC01564=149065,790681,133702
BC01565=149065,790681,133702
BC01566=149065,790681,133702
BC01567=149065,790681,133702
BC01568=117513,790681,53
BC01569=117513,790681,53
BC01570=117513,790681,53
BC01571=117513,790681,53
BC01572=117513,790681,53
BC01573=117513,790681,53
BC01574=117513,790681,53
BC01575=117513,790681,53
BC01576=117513,790681,53
BC01577=117513,790681,53
BC01578=117513,790681,53
BC01579=117513,790681,53
BC01580=117513,790681,53
BC01581=190612,790681,158488
BC01582=190612,790681,158488
BC01583=190612,790681,158488
BC01584=190612,790681,158488
BC01585=190612,790681,158488
BC01586=190612,790681,158488
BC01587=184906,790681,111068
BC01588=184906,790681,111068
BC01589=184906,790681,111068
BC01590=184906,790681,111068
BC01591=184906,790681,111068
BC01592=184906,790681,111068
BC01593=181347,790681,153019
BC01594=174520,790681,233505
BC01595=174520,790681,233505
BC01596=174520,790681,233505
BC01597=174520,790681,233505
BC01598=174520,790681,233505
BC01599=174520,790681,233505
BC01600=184991,733498,315883
BC01601=196160,672502,403752
BC01602=196160,672502,403752
BC01603=237635,668196,305769
BC01604=308625,748445,196549
BC01605=309549,790681,184299
BC01606=309549,790681,184299
BC01607=309549,790681,184299
BC01608=309549,790681,184299
BC01609=309549,790681,184299
BC01610=309549,790681,184299
BC01611=321199,790681,207159
BC01612=321199,790681,207159
BC01613=321199,790681,207159
BC01614=321199,790681,207159
BC01615=321199,790681,207159
BC01616=321199,790681,207159
BC01617=321199,790681,207159
BC01618=321199,790681,207159
BC01619=373020,790681,107875
BC01620=373020,790681,107875
BC01621=373020,790681,107875
BC01622=373020,790681,107875
BC01623=373020,790681,107875
BC01624=373020,790681,107875
BC01625=373020,790681,107875
BC01626=373020,790681,107875
BC01627=367447,763418,217217
BC01628=362764,784495,185132
BC01629=361390,790681,53
BC01630=361390,790681,53
BC01631=361390,790681,53
BC01632=361390,790681,53
BC01633=361390,790681,53
BC01634=361390,790681,53
BC01635=340769,790681,53
BC01636=340769,790681,53
BC01637=340769,790681,53
BC01638=340769,790681,53
BC01639=340769,790681,53
BC01640=340769,790681,53
BC01641=340769,790681,53
BC01642=340769,790681,53
BC01643=340769,790681,53
BC01644=340769,790681,53
BC01645=340769,790681,53
BC01646=340769,790681,53
BC01647=340769,790681,53
BC01648=340769,790681,53
BC01649=340769,790681,53
BC01650=340769,765105,53
BC01651=340769,765105,53
BC01652=340769,765105,53
BC01653=340769,765105,53
BC01654=340769,765105,53
BC01655=340769,765105,53
BC01656=340769,765105,53
BC01657=326290,746662,147117
BC01658=300313,667687,410966
BC01659=300313,667687,410966
BC01660=200178,761203,279737
BC01661=168613,790681,238372
BC01662=168613,790681,238372
BC01663=168613,790681,238372
BC01664=168612,790681,238372
BC01665=168613,790681,238372
BC01666=168613,790681,238372
BC01667=187396,785580,192031
BC01668=187396,785580,192031
BC01669=187396,785580,192031
BC01670=187396,785580,192031
BC01671=187396,785580,192031
BC01672=187396,785580,192031
BC01673=200178,761203,279737
BC01674=300313,667687,410966
BC01675=300313,667687,410966
BC01676=326290,746662,147117
BC01677=326023,790681,196549
BC01678=326023,790681,196549
BC01679=326023,790681,196549
BC01680=326023,790681,196549
BC01681=326023,790681,196549
BC01682=326023,790681,196549
BC01683=316509,790681,152288
BC01684=316509,790681,152288
BC01685=316509,790681,152288
BC01686=316509,790681,152288
BC01687=316509,790681,152288
BC01688=316509,790681,152288
BC01689=314401,774670,185962
BC01690=300313,667687,410966
BC01691=300313,667687,410966
BC01692=200178,761203,279737
BC01693=186958,779092,256601
BC01694=178395,790681,241614
BC01695=178395,790681,241614
BC01696=178395,790681,241614
BC01697=178395,790681,241614
BC01698=178395,790681,241614
BC01699=178395,790681,241614
BC01700=198041,770354,161044
BC01701=198041,770354,161044
BC01702=198041,770354,161044
BC01703=198041,770354,161044
BC01704=198041,770354,161044
BC01705=198041,770354,161044
BC01706=200178,761203,279737
BC01707=300313,667687,410966
BC01708=300313,667687,410966
BC01709=363254,767093,179444
BC01710=378190,790681,124507
BC01711=378190,790681,124507
BC01712=378190,790681,124507
BC01713=378190,790681,124507
BC01714=378190,790681,124507
BC01715=378190,790681,124507
BC01716=345239,790681,222063
BC01717=345239,790681,222063
BC01718=345239,790681,222063
BC01719=345239,790681,222063
BC01720=345239,790681,222063
BC01721=345239,790681,222063
BC01722=363254,767093,179444
BC01723=300313,667687,410966
BC01724=300313,667687,410966
BC01725=200178,761203,279737
BC01726=142668,790681,138813
BC01727=142668,790681,138813
BC01728=142668,790681,138813
BC01729=142668,790681,138813
BC01730=142668,790681,138813
BC01731=142668,790681,138813
BC01732=142668,790681,138813
BC01733=142668,790681,138813
BC01734=203164,773756,23252
BC01735=203164,773756,23252
BC01736=203164,773756,23252
BC01737=203164,773756,23252
BC01738=203164,773756,23252
BC01739=203164,773756,23252
BC01740=200599,780936,88057
BC01741=197119,790681,176008
BC01742=197119,790681,176008
BC01743=197119,790681,176008
BC01744=197119,790681,176008
BC01745=197119,790681,176008
BC01746=197119,790681,176008
BC01747=197993,782258,205645
BC01748=199960,763308,272330
BC01749=201592,760202,280395
BC01750=200178,669563,279737
BC01751=78393,670967,1075175
EC00000=798156,0
EC00001=798153,3
EC00002=798156,0
EC00003=798156,0
EC00004=798156,0
EC00005=798156,0
EC00006=798156,0
EC00007=798156,0
EC00008=798156,0
EC00009=798156,0
EC00010=798156,0
EC00011=798156,0
EC00012=798156,0
EC00013=798156,0
EC00014=798156,0
EC00015=798156,0
EC00016=798156,0
EC00017=798156,0
EC00018=798156,0
EC00019=798156,0
EC00020=798156,0
EC00021=798156,0
EC00022=798156,0
EC00023=798156,0
EC00024=798156,0
EC00025=798156,0
EC00026=798156,0
EC00027=798156,0
EC00028=798156,0
EC00029=798156,0
EC00030=798156,0
EC00031=798156,0
EC00032=798156,0
EC00033=798156,0
EC00034=798156,0
EC00035=798156,0
EC00036=798156,0
EC00037=798156,0
EC00038=798156,0
EC00039=798156,0
EC00040=798156,0
EC00041=798156,0
EC00042=798156,0
EC00043=798156,0
EC00044=798156,0
EC00045=798156,0
EC00046=798156,0
EC00047=798156,0
EC00048=798156,0
EC00049=798156,0
EC00050=798156,0
EC00051=798156,0
EC00052=798156,0
EC00053=798156,0
EC00054=798156,0
EC00055=798156,0
EC00056=798156,0
EC00057=798156,0
EC00058=798156,0
EC00059=798156,0
EC00060=798156,0
EC00061=798156,0
EC00062=798156,0
EC00063=798156,0
EC00064=798156,0
EC00065=798156,0
EC00066=798156,0
EC00067=798156,0
EC00068=798156,0
EC00069=798156,0
EC00070=798156,0
EC00071=798156,0
EC00072=798156,0
EC00073=798156,0
EC00074=798156,0
EC00075=798156,0
EC00076=798156,0
EC00077=798156,0
EC00078=798156,0
EC00079=798156,0
EC00080=798156,0
EC00081=798156,0
EC00082=798156,0
EC00083=798156,0
EC00084=798156,0
EC00085=798156,0
EC00086=798156,0
EC00087=798156,0
EC00088=798156,0
EC00089=798156,0
EC00090=798156,0
EC00091=798156,0
EC00092=798156,0
EC00093=798156,0
EC00094=798156,0
EC00095=798156,0
EC00096=798156,0
EC00097=798156,0
EC00098=798156,0
EC00099=798156,0
EC00100=798156,0
EC00101=798156,0
EC00102=798156,0
EC00103=798156,0
EC00104=798156,0
EC00105=798156,0
EC00106=798156,0
EC00107=798156,0
EC00108=798156,0
EC00109=798156,0
EC00110=798156,0
EC00111=798156,0
EC00112=798156,0
EC00113=798156,0
EC00114=798156,0
EC00115=798155,0
EC00116=798155,0
EC00117=798155,0
EC00118=798155,0
EC00119=798155,0
EC00120=798155,0
EC00121=798155,0
EC00122=798155,0
EC00123=798155,0
EC00124=798156,0
EC00125=798156,0
EC00126=798156,0
EC00127=798156,0
EC00128=798156,0
EC00129=798156,0
EC00130=798156,0
EC00131=798156,0
EC00132=798156,0
EC00133=798156,0
EC00134=798156,0
EC00135=798156,0
EC00136=798156,0
EC00137=798156,0
EC00138=798156,0
EC00139=798156,0
EC00140=798156,0
EC00141=798156,0
EC00142=798156,0
EC00143=798156,0
EC00144=798156,0
EC00145=798156,0
EC00146=798156,0
EC00147=798156,0
EC00148=798156,0
EC00149=798156,0
EC00150=798156,0
EC00151=798156,0
EC00152=798156,0
EC00153=798156,0
EC00154=798156,0
EC00155=798156,0
EC00156=798156,0
EC00157=798156,0
EC00158=798156,0
EC00159=798156,0
EC00160=798156,0
EC00161=798156,0
EC00162=798156,0
EC00163=798156,0
EC00164=798156,0
EC00165=798156,0
EC00166=798156,0
EC00167=798156,0
EC00168=798156,0
EC00169=798156,0
EC00170=798156,0
EC00171=798156,0
EC00172=798156,0
EC00173=798156,0
EC00174=798156,0
EC00175=798156,0
EC00176=798156,0
EC00177=798156,0
EC00178=798156,0
EC00179=798156,0
EC00180=798156,0
EC00181=798156,0
EC00182=798156,0
EC00183=798156,0
EC00184=798156,0
EC00185=798156,0
EC00186=798156,0
EC00187=798156,0
EC00188=798156,0
EC00189=798156,0
EC00190=798156,0
EC00191=798156,0
EC00192=798156,0
EC00193=798156,0
EC00194=798156,0
EC00195=798156,0
EC00196=798156,0
EC00197=798156,0
EC00198=798156,0
EC00199=798156,0
EC00200=798156,0
EC00201=798156,0
EC00202=798156,0
EC00203=798156,0
EC00204=798156,0
EC00205=798156,0
EC00206=798156,0
EC00207=798156,0
EC00208=798156,0
EC00209=798156,0
EC00210=798156,0
EC00211=798156,0
EC00212=798156,0
EC00213=798156,0
EC00214=798156,0
EC00215=798156,0
EC00216=798156,0
EC00217=798156,0
EC00218=798156,0
EC00219=798154,2
EC00220=798156,0
EC00221=798156,0
EC00222=798156,0
EC00223=798156,0
EC00224=798156,0
EC00225=798156,0
EC00226=798156,0
EC00227=798156,0
EC00228=798156,0
EC00229=798156,0
EC00230=798156,0
EC00231=798156,0
EC00232=798156,0
EC00233=798156,0
EC00234=798156,0
EC00235=798156,0
EC00236=798156,0
EC00237=798156,0
EC00238=798156,0
EC00239=798156,0
EC00240=798156,0
EC00241=798156,0
EC00242=798156,0
EC00243=798156,0
EC00244=798156,0
EC00245=798156,0
EC00246=798156,0
EC00247=798156,0
EC00248=798156,0
EC00249=798156,0
EC00250=798156,0
EC00251=798156,0
EC00252=798156,0
EC00253=798156,0
EC00254=798156,0
EC00255=798156,0
EC00256=798156,0
EC00257=798156,0
EC00258=798156,0
EC00259=798156,0
EC00260=798156,0
EC00261=798156,0
EC00262=798156,0
EC00263=798156,0
EC00264=798156,0
EC00265=798156,0
EC00266=798156,0
EC00267=798156,0
EC00268=798156,0
EC00269=798156,0
EC00270=798156,0
EC00271=798156,0
EC00272=798156,0
EC00273=798156,0
EC00274=798156,0
EC00275=798156,0
EC00276=798156,0
EC00277=798156,0
EC00278=798156,0
EC00279=798156,0
EC00280=798156,0
EC00281=798156,0
EC00282=798156,0
EC00283=798156,0
EC00284=798156,0
EC00285=798156,0
EC00286=798156,0
EC00287=798156,0
EC00288=798156,0
EC00289=798156,0
EC00290=798156,0
EC00291=798156,0
EC00292=798156,0
EC00293=798156,0
EC00294=798156,0
EC00295=798156,0
EC00296=798156,0
EC00297=798156,0
EC00298=798156,0
EC00299=798156,0
EC00300=798156,0
EC00301=798156,0
EC00302=798156,0
EC00303=798156,0
EC00304=798156,0
EC00305=798156,0
EC00306=798156,0
EC00307=798156,0
EC00308=798156,0
EC00309=798156,0
EC00310=798156,0
EC00311=798156,0
EC00312=798156,0
EC00313=798156,0
EC00314=798156,0
EC00315=798156,0
EC00316=798156,0
EC00317=798156,0
EC00318=798156,0
EC00319=798156,0
EC00320=798156,0
EC00321=798156,0
EC00322=798156,0
EC00323=798156,0
EC00324=798156,0
EC00325=798156,0
EC00326=798156,0
EC00327=798156,0
EC00328=798156,0
EC00329=798156,0
EC00330=798156,0
EC00331=798156,0
EC00332=798156,0
EC00333=798156,0
EC00334=798156,0
EC00335=798156,0
EC00336=798156,0
EC00337=798156,0
EC00338=798156,0
EC00339=798156,0
EC00340=798156,0
EC00341=798156,0
EC00342=798156,0
EC00343=798156,0
EC00344=798156,0
EC00345=798156,0
EC00346=798156,0
EC00347=798156,0
EC00348=798156,0
EC00349=798156,0
EC00350=798156,0
EC00351=798156,0
EC00352=798156,0
EC00353=798156,0
EC00354=798156,0
EC00355=798156,0
EC00356=798156,0
EC00357=798156,0
EC00358=798155,0
EC00359=798155,0
EC00360=798156,0
EC00361=798155,0
EC00362=798156,0
EC00363=798156,0
EC00364=798156,0
EC00365=798156,0
EC00366=798156,0
EC00367=798156,0
EC00368=798156,0
EC00369=798156,0
EC00370=798156,0
EC00371=798156,0
EC00372=798156,0
EC00373=798156,0
EC00374=798156,0
EC00375=798156,0
EC00376=798156,0
EC00377=798156,0
EC00378=798156,0
EC00379=798156,0
EC00380=798156,0
EC00381=798156,0
EC00382=798156,0
EC00383=798156,0
EC00384=798156,0
EC00385=798156,0
EC00386=798156,0
EC00387=798156,0
EC00388=798156,0
EC00389=798156,0
EC00390=798156,0
EC00391=798156,0
EC00392=798156,0
EC00393=798156,0
EC00394=798156,0
EC00395=798156,0
EC00396=798156,0
EC00397=798156,0
EC00398=798156,0
EC00399=798156,0
EC00400=798156,0
EC00401=798156,0
EC00402=798156,0
EC00403=798156,0
EC00404=798156,0
EC00405=798156,0
EC00406=798156,0
EC00407=798156,0
EC00408=798156,0
EC00409=798156,0
EC00410=798156,0
EC00411=798156,0
EC00412=798156,0
EC00413=798156,0
EC00414=798156,0
EC00415=798156,0
EC00416=798156,0
EC00417=798156,0
EC00418=798156,0
EC00419=798156,0
EC00420=798156,0
EC00421=798156,0
EC00422=798156,0
EC00423=798156,0
EC00424=798156,0
EC00425=798156,0
EC00426=798156,0
EC00427=798156,0
EC00428=798156,0
EC00429=798156,0
EC00430=798156,0
EC00431=798156,0
EC00432=798156,0
EC00433=798156,0
EC00434=798156,0
EC00435=798156,0
EC00436=798156,0
EC00437=798156,0
EC00438=798156,0
EC00439=798156,0
EC00440=798156,0
EC00441=798156,0
EC00442=798156,0
EC00443=798156,0
EC00444=798156,0
EC00445=798156,0
EC00446=798156,0
EC00447=798156,0
EC00448=798156,0
EC00449=798156,0
EC00450=798156,0
EC00451=798156,0
EC00452=798156,0
EC00453=798156,0
EC00454=798156,0
EC00455=798156,0
EC00456=798156,0
EC00457=798156,0
EC00458=798156,0
EC00459=798156,0
EC00460=798156,0
EC00461=798156,0
EC00462=798156,0
EC00463=798156,0
EC00464=798156,0
EC00465=798156,0
EC00466=798156,0
EC00467=798156,0
EC00468=798156,0
EC00469=798156,0
EC00470=798156,0
EC00471=798156,0
EC00472=798156,0
EC00473=798156,0
EC00474=798156,0
EC00475=798156,0
EC00476=798156,0
EC00477=798156,0
EC00478=798156,0
EC00479=798156,0
EC00480=798156,0
EC00481=798156,0
EC00482=798156,0
EC00483=798156,0
EC00484=798156,0
EC00485=798156,0
EC00486=798156,0
EC00487=798156,0
EC00488=798156,0
EC00489=798156,0
EC00490=798156,0
EC00491=798156,0
EC00492=798156,0
EC00493=798156,0
EC00494=798156,0
EC00495=798156,0
EC00496=798156,0
EC00497=798156,0
EC00498=798156,0
EC00499=798156,0
EC00500=798156,1
EC00501=798156,0
EC00502=798156,0
EC00503=798156,0
EC00504=798156,0
EC00505=798156,0
EC00506=798156,0
EC00507=798156,0
EC00508=798156,0
EC00509=798156,0
EC00510=798156,0
EC00511=798156,0
EC00512=798156,0
EC00513=798156,0
EC00514=798156,0
EC00515=798156,0
EC00516=798156,0
EC00517=798156,0
EC00518=798156,0
EC00519=798156,0
EC00520=798156,0
EC00521=798156,0
EC00522=798156,0
EC00523=798156,0
EC00524=798156,0
EC00525=798156,0
EC00526=798156,0
EC00527=798156,0
EC00528=798156,0
EC00529=798156,0
EC00530=798156,0
EC00531=798156,0
EC00532=798156,0
EC00533=798156,0
EC00534=798156,0
EC00535=798156,0
EC00536=798156,0
EC00537=798156,0
EC00538=798156,0
EC00539=798156,0
EC00540=798156,0
EC00541=798156,0
EC00542=798156,0
EC00543=798156,0
EC00544=798156,0
EC00545=798156,0
EC00546=798156,0
EC00547=798156,0
EC00548=798156,0
EC00549=798156,0
EC00550=798156,0
EC00551=798156,0
EC00552=798156,0
EC00553=798156,0
EC00554=798156,0
EC00555=798156,0
EC00556=798156,0
EC00557=798156,0
EC00558=798156,0
EC00559=798156,0
EC00560=798156,0
EC00561=798156,0
EC00562=798156,0
EC00563=798156,0
EC00564=798156,0
EC00565=798156,0
EC00566=798156,0
EC00567=798156,0
EC00568=798156,0
EC00569=798156,0
EC00570=798156,0
EC00571=798156,0
EC00572=798156,0
EC00573=798156,0
EC00574=798156,0
EC00575=798156,0
EC00576=798156,0
EC00577=798156,0
EC00578=798156,0
EC00579=798156,0
EC00580=798156,0
EC00581=798156,0
EC00582=798156,0
EC00583=798156,0
EC00584=798156,0
EC00585=798156,0
EC00586=798156,0
EC00587=798156,0
EC00588=798156,0
EC00589=798156,0
EC00590=798156,0
EC00591=798156,0
EC00592=798156,0
EC00593=798156,0
EC00594=798156,0
EC00595=798156,0
EC00596=798156,0
EC00597=798156,0
EC00598=798156,0
EC00599=798156,0
EC00600=798156,0
EC00601=798155,0
EC00602=798156,0
EC00603=798156,0
EC00604=798156,0
EC00605=798156,0
EC00606=798156,0
EC00607=798156,0
EC00608=798156,0
EC00609=798156,0
EC00610=798156,0
EC00611=798156,0
EC00612=798156,0
EC00613=798156,0
EC00614=798156,0
EC00615=798156,0
EC00616=798156,0
EC00617=798156,0
EC00618=798156,0
EC00619=798156,0
EC00620=798156,0
EC00621=798156,0
EC00622=798156,0
EC00623=798156,0
EC00624=798156,0
EC00625=798156,0
EC00626=798156,0
EC00627=798156,0
EC00628=798156,0
EC00629=798156,0
EC00630=798156,0
EC00631=798156,0
EC00632=798156,0
EC00633=798156,0
EC00634=798156,0
EC00635=798156,0
EC00636=798156,0
EC00637=798156,0
EC00638=798156,0
EC00639=798156,0
EC00640=798156,0
EC00641=798156,0
EC00642=798156,0
EC00643=798156,0
EC00644=798156,0
EC00645=798156,0
EC00646=798156,0
EC00647=798156,0
EC00648=798156,0
EC00649=798156,0
EC00650=798156,0
EC00651=798156,0
EC00652=798156,0
EC00653=798156,0
EC00654=798156,0
EC00655=798156,0
EC00656=798153,3
EC00657=798156,0
EC00658=798156,0
EC00659=798156,0
EC00660=798156,0
EC00661=798156,0
EC00662=798156,0
EC00663=798156,0
EC00664=798156,0
EC00665=798156,0
EC00666=798156,0
EC00667=798156,0
EC00668=798156,0
EC00669=798156,0
EC00670=798156,0
EC00671=798156,0
EC00672=798156,0
EC00673=798156,0
EC00674=798156,0
EC00675=798156,0
EC00676=798156,0
EC00677=798154,2
EC00678=798154,2
EC00679=798154,2
EC00680=798154,2
EC00681=798154,2
EC00682=798154,2
EC00683=798154,2
EC00684=798156,0
EC00685=798156,0
EC00686=798156,0
EC00687=798156,0
EC00688=798156,0
EC00689=798156,0
EC00690=798156,0
EC00691=798156,0
EC00692=798156,0
EC00693=798156,0
EC00694=798156,0
EC00695=798156,0
EC00696=798156,0
EC00697=798156,0
EC00698=798156,0
EC00699=798156,0
EC00700=798156,0
EC00701=798156,0
EC00702=798156,0
EC00703=798156,0
EC00704=798156,0
EC00705=798156,0
EC00706=798156,0
EC00707=798156,0
EC00708=798156,0
EC00709=798156,0
EC00710=798156,0
EC00711=798156,0
EC00712=798156,0
EC00713=798156,0
EC00714=798156,0
EC00715=798156,0
EC00716=798156,0
EC00717=798156,0
EC00718=798156,0
EC00719=798156,0
EC00720=798156,0
EC00721=798156,0
EC00722=798156,0
EC00723=798156,0
EC00724=798156,0
EC00725=798156,0
EC00726=798156,0
EC00727=798156,0
EC00728=798156,0
EC00729=798156,0
EC00730=798156,0
EC00731=798156,0
EC00732=798156,0
EC00733=798156,0
EC00734=798156,0
EC00735=798156,0
EC00736=798156,0
EC00737=798156,0
EC00738=798156,0
EC00739=798156,0
EC00740=798156,0
EC00741=798156,0
EC00742=798156,0
EC00743=798156,0
EC00744=798156,0
EC00745=798156,0
EC00746=798156,0
EC00747=798156,0
EC00748=798156,0
EC00749=798156,0
EC00750=798156,0
EC00751=798156,0
EC00752=798156,0
EC00753=798156,0
EC00754=798156,0
EC00755=798156,0
EC00756=798156,0
EC00757=798156,0
EC00758=798156,0
EC00759=798156,0
EC00760=798156,0
EC00761=798156,0
EC00762=798156,0
EC00763=798156,0
EC00764=798156,0
EC00765=798156,0
EC00766=798156,0
EC00767=798156,0
EC00768=798156,0
EC00769=798156,0
EC00770=798156,0
EC00771=798156,0
EC00772=798156,0
EC00773=798156,0
EC00774=798156,0
EC00775=798156,0
EC00776=798156,0
EC00777=798155,0
EC00778=798155,0
EC00779=798155,0
EC00780=798155,0
EC00781=798155,0
EC00782=798155,0
EC00783=798155,0
EC00784=798155,0
EC00785=798155,0
EC00786=798156,0
EC00787=798156,0
EC00788=798156,0
EC00789=798156,0
EC00790=798156,0
EC00791=798156,0
EC00792=798156,0
EC00793=798156,0
EC00794=798156,0
EC00795=798156,0
EC00796=798156,0
EC00797=798156,0
EC00798=798156,0
EC00799=798156,0
EC00800=798156,0
EC00801=798156,0
EC00802=798156,0
EC00803=798156,0
EC00804=798156,0
EC00805=798156,0
EC00806=798156,0
EC00807=798156,0
EC00808=798156,0
EC00809=798156,0
EC00810=798156,0
EC00811=798156,0
EC00812=798156,0
EC00813=798156,0
EC00814=798156,0
EC00815=798156,0
EC00816=798156,0
EC00817=798156,0
EC00818=798156,0
EC00819=798156,0
EC00820=798156,0
EC00821=798156,0
EC00822=798156,0
EC00823=798156,0
EC00824=798156,0
EC00825=798156,0
EC00826=798156,0
EC00827=798156,0
EC00828=798156,0
EC00829=798156,0
EC00830=798156,0
EC00831=798156,0
EC00832=798156,0
EC00833=798156,0
EC00834=798156,0
EC00835=798156,0
EC00836=798156,0
EC00837=798156,0
EC00838=798156,0
EC00839=798156,0
EC00840=798156,0
EC00841=798156,0
EC00842=798156,0
EC00843=798156,0
EC00844=798156,0
EC00845=798156,0
EC00846=798156,0
EC00847=798156,0
EC00848=798156,0
EC00849=798156,0
EC00850=798156,0
EC00851=798156,0
EC00852=798156,0
EC00853=798156,0
EC00854=798156,0
EC00855=798156,0
EC00856=798156,0
EC00857=798156,0
EC00858=798156,0
EC00859=798156,0
EC00860=798156,0
EC00861=798156,0
EC00862=798156,0
EC00863=798156,0
EC00864=798156,0
EC00865=798156,0
EC00866=798156,0
EC00867=798156,0
EC00868=798156,0
EC00869=798156,0
EC00870=798156,0
EC00871=798156,0
EC00872=798156,0
EC00873=798156,0
EC00874=798156,0
EC00875=798156,0
EC00876=798156,0
EC00877=798156,0
EC00878=798156,0
EC00879=798156,0
EC00880=798156,0
EC00881=798156,0
EC00882=798156,0
EC00883=798156,0
EC00884=798156,0
EC00885=798156,0
EC00886=798156,0
EC00887=798156,0
EC00888=798156,0
EC00889=798156,0
EC00890=798156,0
EC00891=798156,0
EC00892=798156,0
EC00893=798156,0
EC00894=798156,0
EC00895=798156,0
EC00896=798156,0
EC00897=798156,0
EC00898=798156,0
EC00899=798156,0
EC00900=798156,0
EC00901=798156,0
EC00902=798156,0
EC00903=798156,0
EC00904=798156,0
EC00905=798154,2
EC00906=798156,0
EC00907=798156,0
EC00908=798156,0
EC00909=798156,0
EC00910=798156,0
EC00911=798156,0
EC00912=798156,0
EC00913=798156,0
EC00914=798156,0
EC00915=798156,0
EC00916=798156,0
EC00917=798156,0
EC00918=798156,0
EC00919=798156,0
EC00920=798156,0
EC00921=798156,0
EC00922=798156,0
EC00923=798156,0
EC00924=798156,0
EC00925=798156,0
EC00926=798156,0
EC00927=798156,0
EC00928=798156,0
EC00929=798156,0
EC00930=798156,0
EC00931=798156,0
EC00932=798156,0
EC00933=798156,0
EC00934=798156,0
EC00935=798156,0
EC00936=798156,0
EC00937=798156,0
EC00938=798156,0
EC00939=798156,0
EC00940=798156,0
EC00941=798156,0
EC00942=798156,0
EC00943=798156,0
EC00944=798156,0
EC00945=798156,0
EC00946=798156,0
EC00947=798156,0
EC00948=798156,0
EC00949=798156,0
EC00950=798156,0
EC00951=798156,0
EC00952=798156,0
EC00953=798156,0
EC00954=798156,0
EC00955=798156,0
EC00956=798156,0
EC00957=798156,0
EC00958=798156,0
EC00959=798156,0
EC00960=798156,0
EC00961=798156,0
EC00962=798156,0
EC00963=798156,0
EC00964=798156,0
EC00965=798156,0
EC00966=798156,0
EC00967=798156,0
EC00968=798156,0
EC00969=798156,0
EC00970=798156,0
EC00971=798156,0
EC00972=798156,0
EC00973=798156,0
EC00974=798156,0
EC00975=798156,0
EC00976=798156,0
EC00977=798156,0
EC00978=798156,0
EC00979=798156,0
EC00980=798156,0
EC00981=798156,0
EC00982=798156,0
EC00983=798156,0
EC00984=798156,0
EC00985=798156,0
EC00986=798156,0
EC00987=798156,0
EC00988=798156,0
EC00989=798156,0
EC00990=798156,0
EC00991=798156,0
EC00992=798156,0
EC00993=798156,0
EC00994=798156,0
EC00995=798156,0
EC00996=798156,0
EC00997=798156,0
EC00998=798156,0
EC00999=798156,0
EC01000=798156,0
EC01001=798156,0
EC01002=798156,0
EC01003=798156,0
EC01004=798156,0
EC01005=798156,0
EC01006=798156,0
EC01007=798156,0
EC01008=798156,0
EC01009=798156,0
EC01010=798156,0
EC01011=798156,0
EC01012=798156,0
EC01013=798156,0
EC01014=798156,0
EC01015=798156,0
EC01016=798156,0
EC01017=798156,0
EC01018=798156,0
EC01019=798156,0
EC01020=798156,0
EC01021=798156,0
EC01022=798156,0
EC01023=798156,0
EC01024=798156,0
EC01025=798156,0
EC01026=798156,0
EC01027=798156,0
EC01028=798156,0
EC01029=798156,0
EC01030=798156,0
EC01031=798156,0
EC01032=798156,0
EC01033=798156,0
EC01034=798156,0
EC01035=798156,0
EC01036=798156,0
EC01037=798156,0
EC01038=798156,0
EC01039=798156,0
EC01040=798156,0
EC01041=798156,0
EC01042=798156,0
EC01043=798140,8
EC01044=798155,0
EC01045=798156,0
EC01046=798156,0
EC01047=798156,0
EC01048=798156,0
EC01049=798154,0
EC01050=798154,0
EC01051=798156,0
EC01052=798156,0
EC01053=798156,0
EC01054=798156,0
EC01055=798156,0
EC01056=798156,0
EC01057=798156,0
EC01058=798156,0
EC01059=798156,0
EC01060=798156,0
EC01061=798156,0
EC01062=798156,0
EC01063=798156,0
EC01064=798156,0
EC01065=798156,0
EC01066=798156,0
EC01067=798156,0
EC01068=798156,0
EC01069=798156,0
EC01070=798156,0
EC01071=798156,0
EC01072=798156,0
EC01073=798156,0
EC01074=798156,0
EC01075=798156,0
EC01076=798156,0
EC01077=798155,0
EC01078=798155,0
EC01079=798156,0
EC01080=798155,0
EC01081=798156,0
EC01082=798156,0
EC01083=798156,0
EC01084=798156,0
EC01085=798156,0
EC01086=798156,0
EC01087=798156,0
EC01088=798156,0
EC01089=798156,0
EC01090=798156,0
EC01091=798156,0
EC01092=798156,0
EC01093=798156,0
EC01094=798156,0
EC01095=798156,0
EC01096=798156,0
EC01097=798156,0
EC01098=798156,0
EC01099=798156,0
EC01100=798156,0
EC01101=798156,0
EC01102=798156,0
EC01103=798156,0
EC01104=798156,0
EC01105=798156,0
EC01106=798156,0
EC01107=798156,0
EC01108=798156,0
EC01109=798156,0
EC01110=798156,0
EC01111=798156,0
EC01112=798156,0
EC01113=798156,0
EC01114=798156,0
EC01115=798156,0
EC01116=798156,0
EC01117=798156,0
EC01118=798156,0
EC01119=798156,0
EC01120=798156,0
EC01121=798156,0
EC01122=798156,0
EC01123=798156,0
EC01124=798156,0
EC01125=798156,0
EC01126=798156,0
EC01127=798156,0
EC01128=798156,0
EC01129=798154,1
EC01130=798154,1
EC01131=798154,1
EC01132=798154,1
EC01133=798151,2
EC01134=798156,0
EC01135=798156,0
EC01136=798156,0
EC01137=798156,0
EC01138=798156,0
EC01139=798156,0
EC01140=798156,0
EC01141=798156,0
EC01142=798156,0
EC01143=798156,0
EC01144=798156,0
EC01145=798156,0
EC01146=798156,0
EC01147=798156,0
EC01148=798156,0
EC01149=798156,0
EC01150=798156,0
EC01151=798156,0
EC01152=798156,0
EC01153=798156,0
EC01154=798156,0
EC01155=798156,0
EC01156=798156,0
EC01157=798156,0
EC01158=798156,0
EC01159=798156,0
EC01160=798156,0
EC01161=798156,0
EC01162=798156,0
EC01163=798156,0
EC01164=798156,0
EC01165=798156,0
EC01166=798156,0
EC01167=798156,0
EC01168=798156,0
EC01169=798156,0
EC01170=798156,0
EC01171=798156,0
EC01172=798156,0
EC01173=798156,0
EC01174=798156,0
EC01175=798156,0
EC01176=798156,0
EC01177=798156,0
EC01178=798156,0
EC01179=798156,0
EC01180=798156,0
EC01181=798156,0
EC01182=798156,0
EC01183=798156,0
EC01184=798156,0
EC01185=798156,0
EC01186=798156,0
EC01187=798156,0
EC01188=798156,0
EC01189=798156,0
EC01190=798156,0
EC01191=798156,0
EC01192=798156,0
EC01193=798156,0
EC01194=798156,0
EC01195=798156,0
EC01196=798156,0
EC01197=798156,0
EC01198=798156,0
EC01199=798156,0
EC01200=798156,0
EC01201=798156,0
EC01202=798156,0
EC01203=798156,0
EC01204=798156,0
EC01205=798156,0
EC01206=798156,0
EC01207=798156,0
EC01208=798156,0
EC01209=798156,0
EC01210=798156,0
EC01211=798156,0
EC01212=798156,0
EC01213=798156,0
EC01214=798156,0
EC01215=798156,0
EC01216=798156,0
EC01217=798156,0
EC01218=798156,0
EC01219=798156,0
EC01220=798156,0
EC01221=798156,0
EC01222=798156,0
EC01223=798156,0
EC01224=798156,0
EC01225=798156,0
EC01226=798156,0
EC01227=798156,0
EC01228=798156,1
EC01229=798156,0
EC01230=798156,0
EC01231=798156,0
EC01232=798156,0
EC01233=798156,0
EC01234=798156,0
EC01235=798156,0
EC01236=798156,0
EC01237=798156,0
EC01238=798156,0
EC01239=798156,0
EC01240=798156,0
EC01241=798156,0
EC01242=798156,0
EC01243=798156,0
EC01244=798156,0
EC01245=798156,0
EC01246=798156,0
EC01247=798156,0
EC01248=798156,0
EC01249=798156,0
EC01250=798156,0
EC01251=798156,0
EC01252=798156,0
EC01253=798156,0
EC01254=798156,0
EC01255=798156,0
EC01256=798156,0
EC01257=798156,0
EC01258=798156,0
EC01259=798156,0
EC01260=798156,0
EC01261=798156,0
EC01262=798156,0
EC01263=798156,0
EC01264=798156,0
EC01265=798156,0
EC01266=798156,0
EC01267=798156,0
EC01268=798156,0
EC01269=798156,0
EC01270=798156,0
EC01271=798156,0
EC01272=798156,0
EC01273=798156,0
EC01274=798156,0
EC01275=798156,0
EC01276=798156,0
EC01277=798156,0
EC01278=798156,0
EC01279=798156,0
EC01280=798156,0
EC01281=798156,0
EC01282=798156,0
EC01283=798156,0
EC01284=798156,0
EC01285=798156,0
EC01286=798156,0
EC01287=798156,0
EC01288=798156,0
EC01289=798156,0
EC01290=798156,0
EC01291=798156,0
EC01292=798156,0
EC01293=798156,0
EC01294=798156,0
EC01295=798156,0
EC01296=798156,0
EC01297=798156,0
EC01298=798156,0
EC01299=798156,0
EC01300=798156,0
EC01301=798156,0
EC01302=798156,0
EC01303=798156,0
EC01304=798156,0
EC01305=798156,0
EC01306=798156,0
EC01307=798156,0
EC01308=798156,0
EC01309=798156,0
EC01310=798156,0
EC01311=798156,0
EC01312=798156,0
EC01313=798156,0
EC01314=798156,0
EC01315=798156,0
EC01316=798156,0
EC01317=798156,0
EC01318=798156,0
EC01319=798156,0
EC01320=798156,0
EC01321=798155,0
EC01322=798156,0
EC01323=798156,0
EC01324=798156,0
EC01325=798156,0
EC01326=798155,1
EC01327=798155,1
EC01328=798155,1
EC01329=798156,0
EC01330=798156,0
EC01331=798156,0
EC01332=798156,0
EC01333=798156,0
EC01334=798156,0
EC01335=798156,0
EC01336=798156,0
EC01337=798156,0
EC01338=798156,0
EC01339=798156,0
EC01340=798156,0
EC01341=798156,0
EC01342=798156,0
EC01343=798156,0
EC01344=798156,0
EC01345=798156,0
EC01346=798156,0
EC01347=798156,0
EC01348=798156,0
EC01349=798156,0
EC01350=798156,0
EC01351=798156,0
EC01352=798156,0
EC01353=798156,0
EC01354=798156,0
EC01355=798156,0
EC01356=798156,0
EC01357=798156,0
EC01358=798156,0
EC01359=798156,0
EC01360=798156,0
EC01361=798156,0
EC01362=798156,0
EC01363=798156,0
EC01364=798156,0
EC01365=798156,0
EC01366=798155,0
EC01367=798156,0
EC01368=798156,0
EC01369=798156,0
EC01370=798156,0
EC01371=798156,0
EC01372=798156,0
EC01373=798156,0
EC01374=798156,0
EC01375=798156,0
EC01376=798156,0
EC01377=798156,0
EC01378=798156,0
EC01379=798156,0
EC01380=798156,0
EC01381=798156,0
EC01382=798156,0
EC01383=798156,0
EC01384=798156,0
EC01385=798156,0
EC01386=798156,0
EC01387=798156,0
EC01388=798156,0
EC01389=798156,0
EC01390=798156,0
EC01391=798156,0
EC01392=798156,0
EC01393=798156,0
EC01394=798156,0
EC01395=798156,0
EC01396=798156,0
EC01397=798156,0
EC01398=798156,0
EC01399=798156,0
EC01400=798156,0
EC01401=798156,0
EC01402=798156,0
EC01403=798156,0
EC01404=798156,0
EC01405=798156,0
EC01406=798156,0
EC01407=798156,0
EC01408=798156,0
EC01409=798156,0
EC01410=798156,0
EC01411=798156,0
EC01412=798156,0
EC01413=798156,0
EC01414=798156,0
EC01415=798156,0
EC01416=798156,0
EC01417=798156,0
EC01418=798156,0
EC01419=798156,0
EC01420=798156,0
EC01421=798156,0
EC01422=798156,0
EC01423=798156,0
EC01424=798156,0
EC01425=798156,0
EC01426=798153,2
EC01427=798153,2
EC01428=798153,2
EC01429=798153,2
EC01430=798153,2
EC01431=798153,2
EC01432=798153,2
EC01433=798153,2
EC01434=798152,2
EC01435=798152,2
EC01436=798152,2
EC01437=798152,2
EC01438=798152,2
EC01439=798152,2
EC01440=798152,2
EC01441=798153,1
EC01442=798156,0
EC01443=798156,0
EC01444=798156,0
EC01445=798156,0
EC01446=798156,0
EC01447=798156,0
EC01448=798156,0
EC01449=798156,0
EC01450=798156,0
EC01451=798156,0
EC01452=798156,0
EC01453=798156,0
EC01454=798156,0
EC01455=798156,0
EC01456=798156,0
EC01457=798156,0
EC01458=798156,0
EC01459=798156,0
EC01460=798156,0
EC01461=798156,0
EC01462=798156,0
EC01463=798156,0
EC01464=798156,0
EC01465=798156,0
EC01466=798156,0
EC01467=798156,0
EC01468=798156,0
EC01469=798156,0
EC01470=798156,0
EC01471=798156,0
EC01472=798156,0
EC01473=798156,0
EC01474=798154,1
EC01475=798154,1
EC01476=798156,0
EC01477=798156,0
EC01478=798156,0
EC01479=798156,0
EC01480=798156,0
EC01481=798156,0
EC01482=798156,0
EC01483=798156,0
EC01484=798156,0
EC01485=798156,0
EC01486=798156,0
EC01487=798156,0
EC01488=798156,0
EC01489=798156,0
EC01490=798156,0
EC01491=798156,0
EC01492=798156,0
EC01493=798156,0
EC01494=798156,0
EC01495=798156,0
EC01496=798156,0
EC01497=798156,0
EC01498=798156,0
EC01499=798156,0
EC01500=798156,0
EC01501=798156,0
EC01502=798156,0
EC01503=798156,0
EC01504=798156,0
EC01505=798156,1
EC01506=798156,1
EC01507=798156,1
EC01508=798156,1
EC01509=798156,1
EC01510=798156,1
EC01511=798156,1
EC01512=798156,1
EC01513=798156,1
EC01514=798156,1
EC01515=798156,1
EC01516=798156,1
EC01517=798156,1
EC01518=798156,0
EC01519=798156,0
EC01520=798156,0
EC01521=798156,0
EC01522=798156,0
EC01523=798156,0
EC01524=798156,0
EC01525=798156,0
EC01526=798156,0
EC01527=798156,0
EC01528=798156,0
EC01529=798156,0
EC01530=798156,0
EC01531=798156,0
EC01532=798156,0
EC01533=798156,0
EC01534=798156,0
EC01535=798156,0
EC01536=798156,0
EC01537=798156,0
EC01538=798156,0
EC01539=798156,0
EC01540=798156,0
EC01541=798156,0
EC01542=798156,0
EC01543=798156,0
EC01544=798156,0
EC01545=798156,0
EC01546=798156,0
EC01547=798156,0
EC01548=798156,0
EC01549=798156,0
EC01550=798156,0
EC01551=798156,0
EC01552=798156,0
EC01553=798156,0
EC01554=798156,0
EC01555=798156,0
EC01556=798156,0
EC01557=798156,0
EC01558=798156,0
EC01559=798156,0
EC01560=798156,0
EC01561=798156,0
EC01562=798156,0
EC01563=798156,0
EC01564=798156,0
EC01565=798156,0
EC01566=798156,0
EC01567=798156,0
EC01568=798156,0
EC01569=798156,0
EC01570=798156,0
EC01571=798156,0
EC01572=798156,0
EC01573=798156,0
EC01574=798156,0
EC01575=798156,0
EC01576=798156,0
EC01577=798156,0
EC01578=798156,0
EC01579=798156,0
EC01580=798156,0
EC01581=798156,0
EC01582=798156,0
EC01583=798156,0
EC01584=798156,0
EC01585=798156,0
EC01586=798156,0
EC01587=798156,0
EC01588=798156,0
EC01589=798156,0
EC01590=798156,0
EC01591=798156,0
EC01592=798156,0
EC01593=798156,0
EC01594=798156,0
EC01595=798156,0
EC01596=798156,0
EC01597=798156,0
EC01598=798156,0
EC01599=798156,0
EC01600=798156,0
EC01601=798156,0
EC01602=798156,0
EC01603=798156,0
EC01604=798156,0
EC01605=798156,0
EC01606=798156,0
EC01607=798156,0
EC01608=798156,0
EC01609=798156,0
EC01610=798156,0
EC01611=798156,0
EC01612=798156,0
EC01613=798156,0
EC01614=798156,0
EC01615=798156,0
EC01616=798156,0
EC01617=798156,0
EC01618=798156,0
EC01619=798156,0
EC01620=798156,0
EC01621=798156,0
EC01622=798156,0
EC01623=798156,0
EC01624=798156,0
EC01625=798156,0
EC01626=798156,0
EC01627=798156,0
EC01628=798156,0
EC01629=798156,0
EC01630=798156,0
EC01631=798156,0
EC01632=798156,0
EC01633=798156,0
EC01634=798156,0
EC01635=798156,0
EC01636=798156,0
EC01637=798156,0
EC01638=798156,0
EC01639=798156,0
EC01640=798156,0
EC01641=798156,0
EC01642=798156,0
EC01643=798156,0
EC01644=798156,0
EC01645=798156,0
EC01646=798156,0
EC01647=798156,0
EC01648=798156,0
EC01649=798156,0
EC01650=798156,0
EC01651=798156,0
EC01652=798156,0
EC01653=798156,0
EC01654=798156,0
EC01655=798156,0
EC01656=798156,0
EC01657=798156,0
EC01658=798156,0
EC01659=798156,0
EC01660=798156,0
EC01661=798156,0
EC01662=798156,0
EC01663=798156,0
EC01664=798156,0
EC01665=798156,0
EC01666=798156,0
EC01667=798156,0
EC01668=798156,0
EC01669=798156,0
EC01670=798156,0
EC01671=798156,0
EC01672=798156,0
EC01673=798156,0
EC01674=798156,0
EC01675=798156,0
EC01676=798156,0
EC01677=798156,0
EC01678=798156,0
EC01679=798156,0
EC01680=798156,0
EC01681=798156,0
EC01682=798156,0
EC01683=798156,0
EC01684=798156,0
EC01685=798156,0
EC01686=798156,0
EC01687=798156,0
EC01688=798156,0
EC01689=798156,0
EC01690=798156,0
EC01691=798156,0
EC01692=798156,0
EC01693=798156,0
EC01694=798156,0
EC01695=798156,0
EC01696=798156,0
EC01697=798156,0
EC01698=798156,0
EC01699=798156,0
EC01700=798156,0
EC01701=798156,0
EC01702=798156,0
EC01703=798156,0
EC01704=798156,0
EC01705=798156,0
EC01706=798156,0
EC01707=798156,0
EC01708=798156,0
EC01709=798156,0
EC01710=798156,0
EC01711=798156,0
EC01712=798156,0
EC01713=798156,0
EC01714=798156,0
EC01715=798156,0
EC01716=798156,0
EC01717=798156,0
EC01718=798156,0
EC01719=798156,0
EC01720=798156,0
EC01721=798156,0
EC01722=798156,0
EC01723=798156,0
EC01724=798156,0
EC01725=798156,0
EC01726=798156,0
EC01727=798156,0
EC01728=798156,0
EC01729=798156,0
EC01730=798156,0
EC01731=798156,0
EC01732=798156,0
EC01733=798156,0
EC01734=798156,0
EC01735=798156,0
EC01736=798156,0
EC01737=798156,0
EC01738=798156,0
EC01739=798156,0
EC01740=798156,0
EC01741=798156,0
EC01742=798156,0
EC01743=798156,0
EC01744=798156,0
EC01745=798156,0
EC01746=798156,0
EC01747=798156,0
EC01748=798156,0
EC01749=798156,0
EC01750=798156,0
EC01751=798156,0
///POSTYPE BASE
///RECTAN
///RCONF 0,0,0,0,0,0,0,0,0,0,0,0,0,0,0,0,0,0,0,0,0,0,0,0
P00006=0.222,-3.123,-1.508,0.0000,0.0000,0.0000
P00021=-0.225,-6.128,-0.405,0.0000,0.0000,0.0000
P00022=0.222,-3.123,-1.508,0.0000,0.0000,0.0000
P00023=0.143,-0.036,0.682,0.0000,0.0000,0.0000
P00024=0.145,-0.552,1.326,0.0000,0.0000,0.0000
P00025=-2.003,0.006,0.728,0.0000,0.0000,0.0000
P00026=0.562,-0.002,-0.337,0.0000,0.0000,0.0000
P00027=-0.746,0.015,-9.096,0.0000,0.0000,0.0000
P00028=-2.237,-0.018,-7.702,0.0000,0.0000,0.0000
P00029=-2.156,-0.086,-4.681,0.0000,0.0000,0.0000
P00030=5.926,-4.294,-1.390,0.0000,0.0000,0.0000
P00031=1.853,-0.001,-1.549,0.0000,0.0000,0.0000
P00032=1.957,0.503,-7.217,0.0000,0.0000,0.0000
///RCONF 0,0,0,0,1,0,0,0,0,0,0,0,0,0,0,0,0,0,0,0,0,0,0,0
P00033=-0.123,0.612,-5.012,0.0000,0.0000,0.0000
///RCONF 0,0,0,0,0,0,0,0,0,0,0,0,0,0,0,0,0,0,0,0,0,0,0,0
P00034=-0.304,0.773,-2.693,0.0000,0.0000,0.0000
P00035=2.817,0.591,-1.622,0.0000,0.0000,0.0000
P00040=-0.030,9.648,2.467,0.0000,0.0000,0.0000
P00041=0.192,3.924,0.305,0.0000,0.0000,0.0000
P00042=-0.217,1.941,0.413,0.0000,0.0000,0.0000
P00043=-0.044,-1.937,1.197,0.0000,0.0000,0.0000
P00044=0.687,-2.322,1.156,0.0000,0.0000,0.0000
P00045=-0.068,-0.810,1.603,0.0000,0.0000,0.0000
P00046=0.799,0.043,1.292,0.0000,0.0000,0.0000
///RCONF 0,1,0,0,0,0,0,0,0,0,0,0,0,0,0,0,0,0,0,0,0,0,0,0
P00047=-0.011,1.737,-0.646,0.0000,0.0000,0.0000
///RCONF 0,0,0,0,0,0,0,0,0,0,0,0,0,0,0,0,0,0,0,0,0,0,0,0
P00048=2.411,0.025,-0.606,0.0000,0.0000,0.0000
P00049=3.413,-3.572,-1.618,0.0000,0.0000,0.0000
P00050=4.296,-4.501,-0.826,0.0000,0.0000,0.0000
P00051=0.367,3.892,0.009,0.0000,0.0000,0.0000
P00052=0.088,2.832,-0.342,0.0000,0.0000,0.0000
P00053=0.134,6.594,0.107,0.0000,0.0000,0.0000
P00054=-0.103,6.509,-0.702,0.0000,0.0000,0.0000
P00055=-0.342,8.912,1.324,0.0000,0.0000,0.0000
P00061=1.575,-3.405,-0.752,0.0000,0.0000,0.0000
P00062=-0.135,-0.848,-1.706,0.0000,0.0000,0.0000
P00063=0.036,-0.654,-3.005,0.0000,0.0000,0.0000
P00069=2.004,-0.013,0.498,0.0000,0.0000,0.0000
P00071=2.716,0.070,1.352,0.0000,0.0000,0.0000
P00072=1.041,-0.003,-0.797,0.0000,0.0000,0.0000
P00073=-0.961,5.319,-6.157,0.0000,0.0000,0.0000
P00074=1.123,1.944,-5.914,0.0000,0.0000,0.0000
P00080=-3.893,-3.240,-0.208,0.0000,0.0000,0.0000
P00081=19.486,11.347,1.262,0.0000,0.0000,0.0000
P00095=-3.945,4.918,-0.177,0.0000,0.0000,0.0000
P00096=-0.633,5.398,-3.809,0.0000,0.0000,0.0000
P00097=0.069,0.776,0.128,0.0000,0.0000,0.0000
P00098=0.276,2.477,1.230,0.0000,0.0000,0.0000
//INST
///DATE 2025/03/11 13:33
///ATTR SC,RW
///GROUP1 RB1,BS1
///GROUP2 ST1
NOP
COMM 'X2_8A-21A(90,0)
COMM MOVJ C00000 BC00000 VJ=100.00  +MOVJ EC00000 VJ=100.00
COMM CALL JOB:CLEAN-R1_KM_NEW
COMM MOVJ C00001 BC00001 VJ=100.00  +MOVJ EC00001 VJ=100.00
COMM MOVJ C00002 BC00002 VJ=100.00  +MOVJ EC00002 VJ=100.00
COMM 'Path S3463
COMM SFTOF3D
COMM MOVJ C00003 BC00003 VJ=100.00  +MOVJ EC00003 VJ=100.00
COMM MOVL C00004 BC00004 V=666.7  +MOVJ EC00004 VJ=100.00
COMM SMOVL C00005 BC00005 V=166.7  +MOVJ EC00005
COMM SREFP 3 C00006 BC00006  +REFP EC00006
COMM CALL JOB:SEARCH-R1-S13D
COMM SET P095 P006
COMM SFTON3D P095
COMM SMOVL C00007 BC00007 V=166.7  +MOVJ EC00007
COMM SMOVL C00008 BC00008 V=166.7  +MOVJ EC00008
COMM SREFP 3 C00009 BC00009  +REFP EC00009
COMM CALL JOB:SEARCH-R1-S13D
COMM SET P095 P006
COMM SFTON3D P095
COMM SMOVL C00010 BC00010 V=166.7  +MOVJ EC00010
COMM MOVL C00011 BC00011 V=1000.0  +MOVJ EC00011 VJ=100.00
COMM 'EndPath S3463
COMM 'Path S3464
COMM SFTOF3D
COMM MOVJ C00012 BC00012 VJ=100.00  +MOVJ EC00012 VJ=100.00
COMM MOVL C00013 BC00013 V=666.7  +MOVJ EC00013 VJ=100.00
COMM SMOVL C00014 BC00014 V=166.7  +MOVJ EC00014
COMM SREFP 3 C00015 BC00015  +REFP EC00015
COMM CALL JOB:SEARCH-R1-S13D
COMM SET P096 P006
COMM SFTON3D P096
COMM SMOVL C00016 BC00016 V=166.7  +MOVJ EC00016
COMM SREFP 3 C00017 BC00017  +REFP EC00017
COMM CALL JOB:SEARCH-R1-S13D
COMM SET P096 P006
COMM SFTON3D P096
COMM SMOVL C00018 BC00018 V=166.7  +MOVJ EC00018
COMM MOVL C00019 BC00019 V=1000.0  +MOVJ EC00019 VJ=100.00
COMM 'EndPath S3464
COMM 'Path S3465
COMM SFTOF3D
COMM MOVJ C00020 BC00020 VJ=100.00  +MOVJ EC00020 VJ=100.00
COMM MOVL C00021 BC00021 V=666.7  +MOVJ EC00021 VJ=100.00
COMM SMOVL C00022 BC00022 V=166.7  +MOVJ EC00022
COMM SREFP 3 C00023 BC00023  +REFP EC00023
COMM CALL JOB:SEARCH-R1-S13D
COMM SET P021 P006
COMM SFTON3D P021
COMM SMOVL C00024 BC00024 V=166.7  +MOVJ EC00024
COMM SMOVL C00025 BC00025 V=166.7  +MOVJ EC00025
COMM SREFP 3 C00026 BC00026  +REFP EC00026
COMM CALL JOB:SEARCH-R1-S13D
COMM SET P021 P006
COMM SFTON3D P021
COMM SMOVL C00027 BC00027 V=166.7  +MOVJ EC00027
COMM MOVL C00028 BC00028 V=1000.0  +MOVJ EC00028 VJ=100.00
COMM 'EndPath S3465
COMM 'Path S3464
COMM SFTOF3D
COMM MOVJ C00029 BC00029 VJ=100.00  +MOVJ EC00029 VJ=100.00
COMM MOVL C00030 BC00030 V=666.7  +MOVJ EC00030 VJ=100.00
COMM SMOVL C00031 BC00031 V=166.7  +MOVJ EC00031
COMM SREFP 3 C00032 BC00032  +REFP EC00032
COMM CALL JOB:SEARCH-R1-S13D
COMM SET P022 P006
COMM SFTON3D P022
COMM SMOVL C00033 BC00033 V=166.7  +MOVJ EC00033
COMM SREFP 3 C00034 BC00034  +REFP EC00034
COMM CALL JOB:SEARCH-R1-S13D
COMM SET P022 P006
COMM SFTON3D P022
COMM SMOVL C00035 BC00035 V=166.7  +MOVJ EC00035
COMM MOVL C00036 BC00036 V=1000.0  +MOVJ EC00036 VJ=100.00
COMM 'EndPath S3464
COMM MOVJ C00037 BC00037 VJ=100.00  +MOVJ EC00037 VJ=100.00
COMM 'Path S3465
COMM SFTOF3D
COMM MOVJ C00038 BC00038 VJ=100.00  +MOVJ EC00038 VJ=100.00
COMM MOVL C00039 BC00039 V=666.7  +MOVJ EC00039 VJ=100.00
COMM SMOVL C00040 BC00040 V=166.7  +MOVJ EC00040
COMM SREFP 3 C00041 BC00041  +REFP EC00041
COMM CALL JOB:SEARCH-R1-S13D
COMM SET P050 P006
COMM SFTON3D P050
COMM SMOVL C00042 BC00042 V=166.7  +MOVJ EC00042
COMM SREFP 3 C00043 BC00043  +REFP EC00043
COMM CALL JOB:SEARCH-R1-S13D
COMM SET P050 P006
COMM SFTON3D P050
COMM SMOVL C00044 BC00044 V=166.7  +MOVJ EC00044
COMM SMOVL C00045 BC00045 V=166.7  +MOVJ EC00045
COMM SREFP 3 C00046 BC00046  +REFP EC00046
COMM CALL JOB:SEARCH-R1-S13D
COMM SET P050 P006
COMM SFTON3D P050
COMM SMOVL C00047 BC00047 V=166.7  +MOVJ EC00047
COMM MOVL C00048 BC00048 V=1000.0  +MOVJ EC00048 VJ=100.00
COMM 'EndPath S3465
COMM 'Path S3466
COMM SFTOF3D
COMM MOVJ C00049 BC00049 VJ=100.00  +MOVJ EC00049 VJ=100.00
COMM MOVL C00050 BC00050 V=666.7  +MOVJ EC00050 VJ=100.00
COMM SMOVL C00051 BC00051 V=166.7  +MOVJ EC00051
COMM SREFP 3 C00052 BC00052  +REFP EC00052
COMM CALL JOB:SEARCH-R1-S13D
COMM SET P051 P006
COMM SFTON3D P051
COMM SMOVL C00053 BC00053 V=166.7  +MOVJ EC00053
COMM SREFP 3 C00054 BC00054  +REFP EC00054
COMM CALL JOB:SEARCH-R1-S13D
COMM SET P051 P006
COMM SFTON3D P051
COMM SMOVL C00055 BC00055 V=166.7  +MOVJ EC00055
COMM SMOVL C00056 BC00056 V=250.0  +MOVJ EC00056
COMM SREFP 3 C00057 BC00057  +REFP EC00057
COMM CALL JOB:SEARCH-R1-S13D
COMM SET P051 P006
COMM SFTON3D P051
COMM SMOVL C00058 BC00058 V=166.7  +MOVJ EC00058
COMM MOVL C00059 BC00059 V=1000.0  +MOVJ EC00059 VJ=100.00
COMM 'EndPath S3466
COMM MOVJ C00060 BC00060 VJ=100.00  +MOVJ EC00060 VJ=100.00
COMM MOVJ C00061 BC00061 VJ=100.00  +MOVJ EC00061 VJ=100.00
COMM 'Path S3467
COMM SFTOF3D
COMM MOVJ C00062 BC00062 VJ=100.00  +MOVJ EC00062 VJ=100.00
COMM MOVL C00063 BC00063 V=666.7  +MOVJ EC00063 VJ=100.00
COMM SMOVL C00064 BC00064 V=166.7  +MOVJ EC00064
COMM SREFP 3 C00065 BC00065  +REFP EC00065
COMM CALL JOB:SEARCH-R1-S13D
COMM SET P054 P006
COMM SFTON3D P054
COMM SMOVL C00066 BC00066 V=250.0  +MOVJ EC00066
COMM SMOVL C00067 BC00067 V=166.7  +MOVJ EC00067
COMM SREFP 3 C00068 BC00068  +REFP EC00068
COMM CALL JOB:SEARCH-R1-S13D
COMM SET P054 P006
COMM SFTON3D P054
COMM SMOVL C00069 BC00069 V=166.7  +MOVJ EC00069
COMM SMOVL C00070 BC00070 V=800.0  +MOVJ EC00070
COMM SMOVL C00071 BC00071 V=166.7  +MOVJ EC00071
COMM SREFP 3 C00072 BC00072  +REFP EC00072
COMM CALL JOB:SEARCH-R1-S13D
COMM SET P054 P006
COMM SFTON3D P054
COMM SMOVL C00073 BC00073 V=166.7  +MOVJ EC00073
COMM MOVL C00074 BC00074 V=1000.0  +MOVJ EC00074 VJ=100.00
COMM 'EndPath S3467
COMM 'Path S3475
COMM SFTOF3D
COMM MOVJ C00075 BC00075 VJ=100.00  +MOVJ EC00075 VJ=100.00
COMM MOVL C00076 BC00076 V=666.7  +MOVJ EC00076 VJ=100.00
COMM SMOVL C00077 BC00077 V=166.7  +MOVJ EC00077
COMM SREFP 3 C00078 BC00078  +REFP EC00078
COMM CALL JOB:SEARCH-R1-S13D
COMM SET P034 P006
COMM SFTON3D P034
COMM SMOVL C00079 BC00079 V=166.7  +MOVJ EC00079
COMM SMOVL C00080 BC00080 V=333.3  +MOVJ EC00080
COMM SMOVL C00081 BC00081 V=166.7  +MOVJ EC00081
COMM SREFP 3 C00082 BC00082  +REFP EC00082
COMM CALL JOB:SEARCH-R1-S13D
COMM SET P034 P006
COMM SFTON3D P034
COMM SMOVL C00083 BC00083 V=166.7  +MOVJ EC00083
COMM SMOVL C00084 BC00084 V=166.7  +MOVJ EC00084
COMM SREFP 3 C00085 BC00085  +REFP EC00085
COMM CALL JOB:SEARCH-R1-S13D
COMM SET P034 P006
COMM SFTON3D P034
COMM SMOVL C00086 BC00086 V=166.7  +MOVJ EC00086
COMM MOVL C00087 BC00087 V=1000.0  +MOVJ EC00087 VJ=100.00
COMM 'EndPath S3475
COMM 'Path S3464
COMM SFTOF3D
COMM MOVJ C00088 BC00088 VJ=100.00  +MOVJ EC00088 VJ=100.00
COMM MOVL C00089 BC00089 V=666.7  +MOVJ EC00089 VJ=100.00
COMM SMOVL C00090 BC00090 V=166.7  +MOVJ EC00090
COMM SREFP 3 C00091 BC00091  +REFP EC00091
COMM CALL JOB:SEARCH-R1-S13D
COMM SET P023 P006
COMM SFTON3D P023
COMM SMOVL C00092 BC00092 V=166.7  +MOVJ EC00092
COMM SMOVL C00093 BC00093 V=500.0  +MOVJ EC00093
COMM SMOVL C00094 BC00094 V=166.7  +MOVJ EC00094
COMM SREFP 3 C00095 BC00095  +REFP EC00095
COMM CALL JOB:SEARCH-R1-S13D
COMM SET P023 P006
COMM SFTON3D P023
COMM SMOVL C00096 BC00096 V=166.7  +MOVJ EC00096
COMM SMOVL C00097 BC00097 V=166.7  +MOVJ EC00097
COMM SREFP 3 C00098 BC00098  +REFP EC00098
COMM CALL JOB:SEARCH-R1-S13D
COMM SET P023 P006
COMM SFTON3D P023
COMM SMOVL C00099 BC00099 V=166.7  +MOVJ EC00099
COMM MOVL C00100 BC00100 V=1000.0  +MOVJ EC00100 VJ=100.00
COMM MOVJ C00101 BC00101 VJ=80.00  +MOVJ EC00101 VJ=80.00
COMM MOVJ C00102 BC00102 VJ=80.00  +MOVJ EC00102 VJ=80.00
COMM SFTOF3D
COMM MOVJ C00103 BC00103 VJ=80.00  +MOVJ EC00103 VJ=80.00
COMM SMOVL C00104 BC00104 V=166.7  +MOVJ EC00104
COMM SREFP 3 C00105 BC00105  +REFP EC00105
COMM CALL JOB:SEARCH-R1-S13D
COMM SET P061 P006
COMM SFTON3D P061
COMM SMOVL C00106 BC00106 V=166.7  +MOVJ EC00106
COMM SREFP 3 C00107 BC00107  +REFP EC00107
COMM CALL JOB:SEARCH-R1-S13D
COMM SET P061 P006
COMM SFTON3D P061
COMM SMOVL C00108 BC00108 V=166.7  +MOVJ EC00108
COMM SFTOF3D
COMM SMOVL C00109 BC00109 V=500.0  +MOVJ EC00109
COMM SMOVL C00110 BC00110 V=166.7  +MOVJ EC00110
COMM SREFP 3 C00111 BC00111  +REFP EC00111
COMM CALL JOB:SEARCH-R1-S13D
COMM SET P062 P006
COMM SFTON3D P062
COMM SMOVL C00112 BC00112 V=166.7  +MOVJ EC00112
COMM SREFP 3 C00113 BC00113  +REFP EC00113
COMM CALL JOB:SEARCH-R1-S13D
COMM SET P062 P006
COMM SFTON3D P062
COMM SMOVL C00114 BC00114 V=166.7  +MOVJ EC00114
COMM SFTOF3D
COMM SMOVL C00115 BC00115 V=500.0  +MOVJ EC00115
COMM SMOVL C00116 BC00116 V=166.7  +MOVJ EC00116
COMM SREFP 3 C00117 BC00117  +REFP EC00117
COMM CALL JOB:SEARCH-R1-S13D
COMM SET P063 P006
COMM SFTON3D P063
COMM SMOVL C00118 BC00118 V=166.7  +MOVJ EC00118
COMM SREFP 3 C00119 BC00119  +REFP EC00119
COMM CALL JOB:SEARCH-R1-S13D
COMM SET P063 P006
COMM SFTON3D P063
COMM SMOVL C00120 BC00120 V=166.7  +MOVJ EC00120
COMM SFTOF3D
COMM SMOVL C00121 BC00121 V=500.0  +MOVJ EC00121
COMM MOVJ C00122 BC00122 VJ=80.00  +MOVJ EC00122 VJ=80.00
COMM MOVJ C00123 BC00123 VJ=80.00  +MOVJ EC00123 VJ=80.00
COMM 'EndPath S3464
COMM MOVJ C00124 BC00124 VJ=100.00  +MOVJ EC00124 VJ=100.00
COMM 'Path S3465
COMM SFTOF3D
COMM MOVJ C00125 BC00125 VJ=100.00  +MOVJ EC00125 VJ=100.00
COMM MOVL C00126 BC00126 V=666.7  +MOVJ EC00126 VJ=100.00
COMM SMOVL C00127 BC00127 V=166.7  +MOVJ EC00127
COMM SREFP 3 C00128 BC00128  +REFP EC00128
COMM CALL JOB:SEARCH-R1-S13D
COMM SET P024 P006
COMM SFTON3D P024
COMM SMOVL C00129 BC00129 V=166.7  +MOVJ EC00129
COMM SREFP 3 C00130 BC00130  +REFP EC00130
COMM CALL JOB:SEARCH-R1-S13D
COMM SET P024 P006
COMM SFTON3D P024
COMM SMOVL C00131 BC00131 V=166.7  +MOVJ EC00131
COMM SMOVL C00132 BC00132 V=166.7  +MOVJ EC00132
COMM SREFP 3 C00133 BC00133  +REFP EC00133
COMM CALL JOB:SEARCH-R1-S13D
COMM SET P024 P006
COMM SFTON3D P024
COMM SMOVL C00134 BC00134 V=166.7  +MOVJ EC00134
COMM MOVL C00135 BC00135 V=1000.0  +MOVJ EC00135 VJ=100.00
COMM 'EndPath S3465
COMM 'Path S3476
COMM SFTOF3D
COMM MOVJ C00136 BC00136 VJ=100.00  +MOVJ EC00136 VJ=100.00
COMM MOVL C00137 BC00137 V=666.7  +MOVJ EC00137 VJ=100.00
COMM SMOVL C00138 BC00138 V=166.7  +MOVJ EC00138
COMM SREFP 3 C00139 BC00139  +REFP EC00139
COMM CALL JOB:SEARCH-R1-S13D
COMM SET P035 P006
COMM SFTON3D P035
COMM SMOVL C00140 BC00140 V=166.7  +MOVJ EC00140
COMM SREFP 3 C00141 BC00141  +REFP EC00141
COMM CALL JOB:SEARCH-R1-S13D
COMM SET P035 P006
COMM SFTON3D P035
COMM SMOVL C00142 BC00142 V=166.7  +MOVJ EC00142
COMM SMOVL C00143 BC00143 V=333.3  +MOVJ EC00143
COMM SMOVL C00144 BC00144 V=166.7  +MOVJ EC00144
COMM SREFP 3 C00145 BC00145  +REFP EC00145
COMM CALL JOB:SEARCH-R1-S13D
COMM SET P035 P006
COMM SFTON3D P035
COMM SMOVL C00146 BC00146 V=166.7  +MOVJ EC00146
COMM MOVL C00147 BC00147 V=1000.0  +MOVJ EC00147 VJ=100.00
COMM 'EndPath S3476
COMM 'Path S3470
COMM SFTOF3D
COMM MOVJ C00148 BC00148 VJ=100.00  +MOVJ EC00148 VJ=100.00
COMM MOVL C00149 BC00149 V=666.7  +MOVJ EC00149 VJ=100.00
COMM SMOVL C00150 BC00150 V=166.7  +MOVJ EC00150
COMM SREFP 3 C00151 BC00151  +REFP EC00151
COMM CALL JOB:SEARCH-R1-S13D
COMM SET P029 P006
COMM SFTON3D P029
COMM SMOVL C00152 BC00152 V=166.7  +MOVJ EC00152
COMM SREFP 3 C00153 BC00153  +REFP EC00153
COMM CALL JOB:SEARCH-R1-S13D
COMM SET P029 P006
COMM SFTON3D P029
COMM SMOVL C00154 BC00154 V=166.7  +MOVJ EC00154
COMM SMOVL C00155 BC00155 V=250.0  +MOVJ EC00155
COMM SMOVL C00156 BC00156 V=166.7  +MOVJ EC00156
COMM SREFP 3 C00157 BC00157  +REFP EC00157
COMM CALL JOB:SEARCH-R1-S13D
COMM SET P029 P006
COMM SFTON3D P029
COMM SMOVL C00158 BC00158 V=166.7  +MOVJ EC00158
COMM MOVL C00159 BC00159 V=1000.0  +MOVJ EC00159 VJ=100.00
COMM 'EndPath S3470
COMM 'Path S4850
COMM SFTOF3D
COMM MOVL C00160 BC00160 V=666.7  +MOVJ EC00160 VJ=100.00
COMM SMOVL C00161 BC00161 V=166.7  +MOVJ EC00161
COMM SREFP 3 C00162 BC00162  +REFP EC00162
COMM CALL JOB:SEARCH-R1-S13D
COMM SET P071 P006
COMM SFTON3D P071
COMM SMOVL C00163 BC00163 V=166.7  +MOVJ EC00163
COMM SREFP 3 C00164 BC00164  +REFP EC00164
COMM CALL JOB:SEARCH-R1-S13D
COMM SET P071 P006
COMM SFTON3D P071
COMM SMOVL C00165 BC00165 V=166.7  +MOVJ EC00165
COMM SMOVL C00166 BC00166 V=166.7  +MOVJ EC00166
COMM SREFP 3 C00167 BC00167  +REFP EC00167
COMM CALL JOB:SEARCH-R1-S13D
COMM SET P071 P006
COMM SFTON3D P071
COMM SMOVL C00168 BC00168 V=166.7  +MOVJ EC00168
COMM MOVL C00169 BC00169 V=1000.0  +MOVJ EC00169 VJ=100.00
COMM 'EndPath S4850
COMM 'Path S4851
COMM SFTOF3D
COMM MOVJ C00170 BC00170 VJ=100.00  +MOVJ EC00170 VJ=100.00
COMM MOVL C00171 BC00171 V=666.7  +MOVJ EC00171 VJ=100.00
COMM SMOVL C00172 BC00172 V=166.7  +MOVJ EC00172
COMM SREFP 3 C00173 BC00173  +REFP EC00173
COMM CALL JOB:SEARCH-R1-S13D
COMM SET P072 P006
COMM SFTON3D P072
COMM SMOVL C00174 BC00174 V=166.7  +MOVJ EC00174
COMM SREFP 3 C00175 BC00175  +REFP EC00175
COMM CALL JOB:SEARCH-R1-S13D
COMM SET P072 P006
COMM SFTON3D P072
COMM SMOVL C00176 BC00176 V=166.7  +MOVJ EC00176
COMM MOVL C00177 BC00177 V=1000.0  +MOVJ EC00177 VJ=100.00
COMM 'EndPath S4851
COMM MOVJ C00178 BC00178 VJ=100.00  +MOVJ EC00178 VJ=100.00
COMM MOVJ C00179 BC00179 VJ=100.00  +MOVJ EC00179 VJ=100.00
COMM 'Path S4852
COMM SFTOF3D
COMM MOVJ C00180 BC00180 VJ=100.00  +MOVJ EC00180 VJ=100.00
COMM MOVL C00181 BC00181 V=666.7  +MOVJ EC00181 VJ=100.00
COMM SMOVL C00182 BC00182 V=166.7  +MOVJ EC00182
COMM SREFP 3 C00183 BC00183  +REFP EC00183
COMM CALL JOB:SEARCH-R1-S13D
COMM SET P073 P006
COMM SFTON3D P073
COMM SMOVL C00184 BC00184 V=166.7  +MOVJ EC00184
COMM SMOVL C00185 BC00185 V=166.7  +MOVJ EC00185
COMM SREFP 3 C00186 BC00186  +REFP EC00186
COMM CALL JOB:SEARCH-R1-S13D
COMM SET P073 P006
COMM SFTON3D P073
COMM SMOVL C00187 BC00187 V=166.7  +MOVJ EC00187
COMM SMOVL C00188 BC00188 V=166.7  +MOVJ EC00188
COMM SREFP 3 C00189 BC00189  +REFP EC00189
COMM CALL JOB:SEARCH-R1-S13D
COMM SET P073 P006
COMM SFTON3D P073
COMM SMOVL C00190 BC00190 V=166.7  +MOVJ EC00190
COMM MOVL C00191 BC00191 V=1000.0  +MOVJ EC00191 VJ=100.00
COMM 'EndPath S4852
COMM MOVJ C00192 BC00192 VJ=100.00  +MOVJ EC00192 VJ=100.00
COMM 'Path S4853
COMM SFTOF3D
COMM MOVJ C00193 BC00193 VJ=100.00  +MOVJ EC00193 VJ=100.00
COMM MOVL C00194 BC00194 V=666.7  +MOVJ EC00194 VJ=100.00
COMM SMOVL C00195 BC00195 V=166.7  +MOVJ EC00195
COMM SREFP 3 C00196 BC00196  +REFP EC00196
COMM CALL JOB:SEARCH-R1-S13D
COMM SET P074 P006
COMM SFTON3D P074
COMM SMOVL C00197 BC00197 V=166.7  +MOVJ EC00197
COMM SREFP 3 C00198 BC00198  +REFP EC00198
COMM CALL JOB:SEARCH-R1-S13D
COMM SET P074 P006
COMM SFTON3D P074
COMM SMOVL C00199 BC00199 V=166.7  +MOVJ EC00199
COMM MOVL C00200 BC00200 V=1000.0  +MOVJ EC00200 VJ=100.00
COMM 'EndPath S4853
COMM 'Path S3467
COMM SFTOF3D
COMM MOVJ C00201 BC00201 VJ=100.00  +MOVJ EC00201 VJ=100.00
COMM MOVJ C00202 BC00202 VJ=100.00  +MOVJ EC00202 VJ=100.00
COMM MOVJ C00203 BC00203 VJ=100.00  +MOVJ EC00203 VJ=100.00
COMM MOVJ C00204 BC00204 VJ=100.00  +MOVJ EC00204 VJ=100.00
COMM MOVL C00205 BC00205 V=666.7  +MOVJ EC00205 VJ=100.00
COMM SMOVL C00206 BC00206 V=166.7  +MOVJ EC00206
COMM SREFP 3 C00207 BC00207  +REFP EC00207
COMM CALL JOB:SEARCH-R1-S13D
COMM SET P026 P006
COMM SFTON3D P026
COMM SMOVL C00208 BC00208 V=166.7  +MOVJ EC00208
COMM SREFP 3 C00209 BC00209  +REFP EC00209
COMM CALL JOB:SEARCH-R1-S13D
COMM SET P026 P006
COMM SFTON3D P026
COMM SMOVL C00210 BC00210 V=166.7  +MOVJ EC00210
COMM SMOVL C00211 BC00211 V=800.0  +MOVJ EC00211
COMM SMOVL C00212 BC00212 V=166.7  +MOVJ EC00212
COMM SREFP 3 C00213 BC00213  +REFP EC00213
COMM CALL JOB:SEARCH-R1-S13D
COMM SET P026 P006
COMM SFTON3D P026
COMM SMOVL C00214 BC00214 V=166.7  +MOVJ EC00214
COMM MOVL C00215 BC00215 V=1000.0  +MOVJ EC00215 VJ=100.00
COMM 'EndPath S3467
COMM MOVJ C00216 BC00216 VJ=100.00  +MOVJ EC00216 VJ=100.00
COMM 'Path S3466
COMM SFTOF3D
COMM MOVJ C00217 BC00217 VJ=100.00  +MOVJ EC00217 VJ=100.00
COMM MOVL C00218 BC00218 V=666.7  +MOVJ EC00218 VJ=100.00
COMM SMOVL C00219 BC00219 V=166.7  +MOVJ EC00219
COMM SREFP 3 C00220 BC00220  +REFP EC00220
COMM CALL JOB:SEARCH-R1-S13D
COMM SET P025 P006
COMM SFTON3D P025
COMM SMOVL C00221 BC00221 V=166.7  +MOVJ EC00221
COMM SMOVL C00222 BC00222 V=166.7  +MOVJ EC00222
COMM SREFP 3 C00223 BC00223  +REFP EC00223
COMM CALL JOB:SEARCH-R1-S13D
COMM SET P025 P006
COMM SFTON3D P025
COMM SMOVL C00224 BC00224 V=166.7  +MOVJ EC00224
COMM SMOVL C00225 BC00225 V=200.0  +MOVJ EC00225
COMM SMOVL C00226 BC00226 V=166.7  +MOVJ EC00226
COMM SREFP 3 C00227 BC00227  +REFP EC00227
COMM CALL JOB:SEARCH-R1-S13D
COMM SET P025 P006
COMM SFTON3D P025
COMM SMOVL C00228 BC00228 V=166.7  +MOVJ EC00228
COMM MOVL C00229 BC00229 V=1000.0  +MOVJ EC00229 VJ=100.00
COMM 'EndPath S3466
COMM MOVJ C00230 BC00230 VJ=100.00  +MOVJ EC00230 VJ=100.00
COMM 'Path S3469
COMM SFTOF3D
COMM MOVJ C00231 BC00231 VJ=100.00  +MOVJ EC00231 VJ=100.00
COMM MOVL C00232 BC00232 V=666.7  +MOVJ EC00232 VJ=100.00
COMM SMOVL C00233 BC00233 V=166.7  +MOVJ EC00233
COMM SREFP 3 C00234 BC00234  +REFP EC00234
COMM CALL JOB:SEARCH-R1-S13D
COMM SET P028 P006
COMM SFTON3D P028
COMM SMOVL C00235 BC00235 V=166.7  +MOVJ EC00235
COMM SREFP 3 C00236 BC00236  +REFP EC00236
COMM CALL JOB:SEARCH-R1-S13D
COMM SET P028 P006
COMM SFTON3D P028
COMM SMOVL C00237 BC00237 V=166.7  +MOVJ EC00237
COMM SMOVL C00238 BC00238 V=333.3  +MOVJ EC00238
COMM SMOVL C00239 BC00239 V=166.7  +MOVJ EC00239
COMM SREFP 3 C00240 BC00240  +REFP EC00240
COMM CALL JOB:SEARCH-R1-S13D
COMM SET P028 P006
COMM SFTON3D P028
COMM SMOVL C00241 BC00241 V=166.7  +MOVJ EC00241
COMM MOVL C00242 BC00242 V=1000.0  +MOVJ EC00242 VJ=100.00
COMM 'EndPath S3469
COMM MOVJ C00243 BC00243 VJ=100.00  +MOVJ EC00243 VJ=100.00
COMM 'Path S3474
COMM SFTOF3D
COMM MOVJ C00244 BC00244 VJ=100.00  +MOVJ EC00244 VJ=100.00
COMM MOVL C00245 BC00245 V=666.7  +MOVJ EC00245 VJ=100.00
COMM SMOVL C00246 BC00246 V=166.7  +MOVJ EC00246
COMM SREFP 3 C00247 BC00247  +REFP EC00247
COMM CALL JOB:SEARCH-R1-S13D
COMM SET P033 P006
COMM SFTON3D P033
COMM SMOVL C00248 BC00248 V=166.7  +MOVJ EC00248
COMM SREFP 3 C00249 BC00249  +REFP EC00249
COMM CALL JOB:SEARCH-R1-S13D
COMM SET P033 P006
COMM SFTON3D P033
COMM SMOVL C00250 BC00250 V=166.7  +MOVJ EC00250
COMM SMOVL C00251 BC00251 V=250.0  +MOVJ EC00251
COMM SMOVL C00252 BC00252 V=166.7  +MOVJ EC00252
COMM SREFP 3 C00253 BC00253  +REFP EC00253
COMM CALL JOB:SEARCH-R1-S13D
COMM SET P033 P006
COMM SFTON3D P033
COMM SMOVL C00254 BC00254 V=166.7  +MOVJ EC00254
COMM MOVL C00255 BC00255 V=1000.0  +MOVJ EC00255 VJ=100.00
COMM 'EndPath S3474
COMM 'Path S3468
COMM SFTOF3D
COMM MOVJ C00256 BC00256 VJ=100.00  +MOVJ EC00256 VJ=100.00
COMM MOVL C00257 BC00257 V=666.7  +MOVJ EC00257 VJ=100.00
COMM SMOVL C00258 BC00258 V=166.7  +MOVJ EC00258
COMM SREFP 3 C00259 BC00259  +REFP EC00259
COMM CALL JOB:SEARCH-R1-S13D
COMM SET P027 P006
COMM SFTON3D P027
COMM SMOVL C00260 BC00260 V=166.7  +MOVJ EC00260
COMM SMOVL C00261 BC00261 V=166.7  +MOVJ EC00261
COMM SREFP 3 C00262 BC00262  +REFP EC00262
COMM CALL JOB:SEARCH-R1-S13D
COMM SET P027 P006
COMM SFTON3D P027
COMM SMOVL C00263 BC00263 V=166.7  +MOVJ EC00263
COMM SMOVL C00264 BC00264 V=166.7  +MOVJ EC00264
COMM SREFP 3 C00265 BC00265  +REFP EC00265
COMM CALL JOB:SEARCH-R1-S13D
COMM SET P027 P006
COMM SFTON3D P027
COMM SMOVL C00266 BC00266 V=166.7  +MOVJ EC00266
COMM MOVL C00267 BC00267 V=1000.0  +MOVJ EC00267 VJ=100.00
COMM 'EndPath S3468
COMM 'Path S3471
COMM SFTOF3D
COMM MOVJ C00268 BC00268 VJ=100.00  +MOVJ EC00268 VJ=100.00
COMM MOVL C00269 BC00269 V=666.7  +MOVJ EC00269 VJ=100.00
COMM SMOVL C00270 BC00270 V=166.7  +MOVJ EC00270
COMM SREFP 3 C00271 BC00271  +REFP EC00271
COMM CALL JOB:SEARCH-R1-S13D
COMM SET P030 P006
COMM SFTON3D P030
COMM SMOVL C00272 BC00272 V=166.7  +MOVJ EC00272
COMM SREFP 3 C00273 BC00273  +REFP EC00273
COMM CALL JOB:SEARCH-R1-S13D
COMM SET P030 P006
COMM SFTON3D P030
COMM SMOVL C00274 BC00274 V=166.7  +MOVJ EC00274
COMM MOVL C00275 BC00275 V=1000.0  +MOVJ EC00275 VJ=100.00
COMM 'EndPath S3471
COMM 'Path S3472
COMM SFTOF3D
COMM MOVJ C00276 BC00276 VJ=100.00  +MOVJ EC00276 VJ=100.00
COMM MOVL C00277 BC00277 V=666.7  +MOVJ EC00277 VJ=100.00
COMM SMOVL C00278 BC00278 V=166.7  +MOVJ EC00278
COMM SREFP 3 C00279 BC00279  +REFP EC00279
COMM CALL JOB:SEARCH-R1-S13D
COMM SET P031 P006
COMM SFTON3D P031
COMM SMOVL C00280 BC00280 V=166.7  +MOVJ EC00280
COMM SREFP 3 C00281 BC00281  +REFP EC00281
COMM CALL JOB:SEARCH-R1-S13D
COMM SET P031 P006
COMM SFTON3D P031
COMM SMOVL C00282 BC00282 V=166.7  +MOVJ EC00282
COMM MOVL C00283 BC00283 V=1000.0  +MOVJ EC00283 VJ=100.00
COMM 'EndPath S3472
COMM MOVJ C00284 BC00284 VJ=100.00  +MOVJ EC00284 VJ=100.00
COMM 'Path S3472
COMM SFTOF3D
COMM MOVJ C00285 BC00285 VJ=100.00  +MOVJ EC00285 VJ=100.00
COMM MOVL C00286 BC00286 V=666.7  +MOVJ EC00286 VJ=100.00
COMM SMOVL C00287 BC00287 V=166.7  +MOVJ EC00287
COMM SREFP 3 C00288 BC00288  +REFP EC00288
COMM CALL JOB:SEARCH-R1-S13D
COMM SET P032 P006
COMM SFTON3D P032
COMM SMOVL C00289 BC00289 V=166.7  +MOVJ EC00289
COMM SREFP 3 C00290 BC00290  +REFP EC00290
COMM CALL JOB:SEARCH-R1-S13D
COMM SET P032 P006
COMM SFTON3D P032
COMM SMOVL C00291 BC00291 V=166.7  +MOVJ EC00291
COMM SMOVL C00292 BC00292 V=133.3  +MOVJ EC00292
COMM SREFP 3 C00293 BC00293  +REFP EC00293
COMM CALL JOB:SEARCH-R1-S13D
COMM SET P032 P006
COMM SFTON3D P032
COMM SMOVL C00294 BC00294 V=166.7  +MOVJ EC00294
COMM MOVL C00295 BC00295 V=1000.0  +MOVJ EC00295 VJ=100.00
COMM 'EndPath S3472
COMM MOVJ C00296 BC00296 VJ=100.00  +MOVJ EC00296 VJ=100.00
COMM 'Path S3477
COMM SFTOF3D
COMM MOVJ C00297 BC00297 VJ=100.00  +MOVJ EC00297 VJ=100.00
COMM SMOVL C00298 BC00298 V=166.7  +MOVJ EC00298
COMM SREFP 3 C00299 BC00299  +REFP EC00299
COMM CALL JOB:SEARCH-R1-S13D
COMM SET P069 P006
COMM SFTON3D P069
COMM SMOVL C00300 BC00300 V=250.0  +MOVJ EC00300
COMM SMOVL C00301 BC00301 V=250.0  +MOVJ EC00301
COMM SMOVL C00302 BC00302 V=166.7  +MOVJ EC00302
COMM SREFP 3 C00303 BC00303  +REFP EC00303
COMM CALL JOB:SEARCH-R1-S13D
COMM SET P069 P006
COMM SFTON3D P069
COMM SMOVL C00304 BC00304 V=166.7  +MOVJ EC00304
COMM SFTOF3D
COMM SMOVL C00305 BC00305 V=666.7  +MOVJ EC00305
COMM MOVL C00306 BC00306 V=666.7  +MOVJ EC00306 VJ=100.00
COMM SMOVL C00307 BC00307 V=166.7  +MOVJ EC00307
COMM SREFP 3 C00308 BC00308  +REFP EC00308
COMM CALL JOB:SEARCH-R1-S13D
COMM SET P052 P006
COMM SFTON3D P052
COMM SMOVL C00309 BC00309 V=166.7  +MOVJ EC00309
COMM SREFP 3 C00310 BC00310  +REFP EC00310
COMM CALL JOB:SEARCH-R1-S13D
COMM SET P052 P006
COMM SFTON3D P052
COMM SMOVL C00311 BC00311 V=166.7  +MOVJ EC00311
COMM MOVL C00312 BC00312 V=1000.0  +MOVJ EC00312 VJ=100.00
COMM 'EndPath S3477
COMM MOVJ C00313 BC00313 VJ=100.00  +MOVJ EC00313 VJ=100.00
COMM 'poprawiÃÂ searcha- nie mialem
COMM 'wyciecia
COMM 'Path S3478
COMM SFTOF3D
COMM MOVJ C00314 BC00314 VJ=100.00  +MOVJ EC00314 VJ=100.00
COMM MOVL C00315 BC00315 V=666.7  +MOVJ EC00315 VJ=100.00
COMM SMOVL C00316 BC00316 V=166.7  +MOVJ EC00316
COMM SREFP 3 C00317 BC00317  +REFP EC00317
COMM CALL JOB:SEARCH-R1-S13D
COMM SET P053 P006
COMM SFTON3D P053
COMM SMOVL C00318 BC00318 V=166.7  +MOVJ EC00318
COMM SREFP 3 C00319 BC00319  +REFP EC00319
COMM CALL JOB:SEARCH-R1-S13D
COMM SET P053 P006
COMM SFTON3D P053
COMM SMOVL C00320 BC00320 V=166.7  +MOVJ EC00320
COMM MOVL C00321 BC00321 V=1000.0  +MOVJ EC00321 VJ=100.00
COMM 'EndPath S3478
COMM '
COMM MOVJ C00322 BC00322 VJ=100.00  +MOVJ EC00322 VJ=100.00
COMM 'Path W3476
COMM SFTOF3D
COMM SFTON3D P033
COMM MOVJ C00323 BC00323 VJ=100.00  +MOVJ EC00323 VJ=100.00
COMM SMOVL C00324 BC00324 V=800.0  +MOVJ EC00324
COMM SMOVL C00325 BC00325 V=166.7 PL=0  +MOVJ EC00325
COMM MACRO1 MJ#(0) ARGF14
COMM ARCON
COMM SMOVL C00326 BC00326 V=10.0  +MOVJ EC00326
COMM ARCOF
COMM SMOVL C00327 BC00327 V=800.0  +MOVJ EC00327
COMM SMOVL C00328 BC00328 V=1000.0  +MOVJ EC00328
COMM SFTOF3D
COMM 'EndPath W3476
COMM 'Path W3477
COMM SFTOF3D
COMM SFTON3D P033
COMM MOVJ C00329 BC00329 VJ=100.00  +MOVJ EC00329 VJ=100.00
COMM SMOVL C00330 BC00330 V=800.0  +MOVJ EC00330
COMM SMOVL C00331 BC00331 V=166.7 PL=0  +MOVJ EC00331
COMM SMOVL C00332 BC00332 V=10.0  +MOVJ EC00332
COMM SMOVL C00333 BC00333 V=10.0  +MOVJ EC00333
COMM SMOVL C00334 BC00334 V=10.0  +MOVJ EC00334
COMM ARCOF
COMM SMOVL C00335 BC00335 V=800.0  +MOVJ EC00335
COMM SMOVL C00336 BC00336 V=1000.0  +MOVJ EC00336
COMM SFTOF3D
COMM 'EndPath W3477
COMM MOVJ C00337 BC00337 VJ=100.00  +MOVJ EC00337 VJ=100.00
COMM 'Path W3478
COMM SFTOF3D
COMM SFTON3D P033
COMM MOVJ C00338 BC00338 VJ=100.00  +MOVJ EC00338 VJ=100.00
COMM SMOVL C00339 BC00339 V=800.0  +MOVJ EC00339
COMM SMOVL C00340 BC00340 V=166.7 PL=0  +MOVJ EC00340
COMM ARCON
COMM SMOVL C00341 BC00341 V=10.0  +MOVJ EC00341
COMM SMOVL C00342 BC00342 V=10.0  +MOVJ EC00342
COMM SMOVL C00343 BC00343 V=10.0  +MOVJ EC00343
COMM ARCOF
COMM SMOVL C00344 BC00344 V=800.0  +MOVJ EC00344
COMM SMOVL C00345 BC00345 V=1000.0  +MOVJ EC00345
COMM SFTOF3D
COMM 'EndPath W3478
COMM MOVJ C00346 BC00346 VJ=100.00  +MOVJ EC00346 VJ=100.00
COMM MOVJ C00347 BC00347 VJ=100.00  +MOVJ EC00347 VJ=100.00
COMM '9
COMM 'Path W3479
COMM SFTOF3D
COMM SFTON3D P026
COMM MOVJ C00348 BC00348 VJ=100.00  +MOVJ EC00348 VJ=100.00
COMM SMOVL C00349 BC00349 V=800.0  +MOVJ EC00349
COMM SMOVL C00350 BC00350 V=166.7 PL=0  +MOVJ EC00350
COMM ARCON
COMM SMOVL C00351 BC00351 V=9.2  +MOVJ EC00351
COMM SMOVL C00352 BC00352 V=9.2  +MOVJ EC00352
COMM SMOVL C00353 BC00353 V=9.2  +MOVJ EC00353
COMM ARCOF
COMM SMOVL C00354 BC00354 V=800.0  +MOVJ EC00354
COMM SMOVL C00355 BC00355 V=1000.0  +MOVJ EC00355
COMM SFTOF3D
COMM 'EndPath W3479
COMM 'Path W3480
COMM SFTOF3D
COMM SFTON3D P026
COMM MOVJ C00356 BC00356 VJ=100.00  +MOVJ EC00356 VJ=100.00
COMM SMOVL C00357 BC00357 V=800.0  +MOVJ EC00357
COMM SMOVL C00358 BC00358 V=150.0 PL=0  +MOVJ EC00358
COMM ARCON
COMM SMOVL C00359 BC00359 V=10.0  +MOVJ EC00359
COMM SMOVL C00360 BC00360 V=10.0  +MOVJ EC00360
COMM SMOVL C00361 BC00361 V=10.0  +MOVJ EC00361
COMM ARCOF
COMM SMOVL C00362 BC00362 V=800.0  +MOVJ EC00362
COMM SMOVL C00363 BC00363 V=1000.0  +MOVJ EC00363
COMM SFTOF3D
COMM 'EndPath W3480
COMM 'Path W3481
COMM SFTOF3D
COMM SFTON3D P026
COMM MOVJ C00364 BC00364 VJ=100.00  +MOVJ EC00364 VJ=100.00
COMM SMOVL C00365 BC00365 V=800.0  +MOVJ EC00365
COMM SMOVL C00366 BC00366 V=150.0 PL=0  +MOVJ EC00366
COMM SMOVL C00367 BC00367 V=10.0  +MOVJ EC00367
COMM ARCOF
COMM SMOVL C00368 BC00368 V=800.0  +MOVJ EC00368
COMM SMOVL C00369 BC00369 V=1000.0  +MOVJ EC00369
COMM SFTOF3D
COMM 'EndPath W3481
COMM MOVJ C00370 BC00370 VJ=100.00  +MOVJ EC00370 VJ=100.00
COMM 'uwaga na podajnik
COMM 'Path W3481
COMM SFTOF3D
COMM SFTON3D P026
COMM MOVJ C00371 BC00371 VJ=50.00  +MOVJ EC00371 VJ=15.00
COMM SMOVL C00372 BC00372 V=800.0  +MOVJ EC00372
COMM SMOVL C00373 BC00373 V=150.0 PL=0  +MOVJ EC00373
COMM ARCON
COMM SMOVL C00374 BC00374 V=10.0  +MOVJ EC00374
COMM SMOVL C00375 BC00375 V=10.0  +MOVJ EC00375
COMM ARCOF
COMM SMOVL C00376 BC00376 V=800.0  +MOVJ EC00376
COMM SMOVL C00377 BC00377 V=1000.0  +MOVJ EC00377
COMM SFTOF3D
COMM 'EndPath W3481
COMM 'brak dostepu offset drutu 1cm
COMM 'Path W3482
COMM SFTOF3D
COMM SFTON3D P026
COMM MOVJ C00378 BC00378 VJ=100.00  +MOVJ EC00378 VJ=100.00
COMM SMOVL C00379 BC00379 V=800.0  +MOVJ EC00379
COMM SMOVL C00380 BC00380 V=150.0 PL=0  +MOVJ EC00380
COMM ARCON
COMM SMOVL C00381 BC00381 V=10.0  +MOVJ EC00381
COMM ARCOF
COMM SMOVL C00382 BC00382 V=800.0  +MOVJ EC00382
COMM SMOVL C00383 BC00383 V=1000.0  +MOVJ EC00383
COMM SFTOF3D
COMM 'EndPath W3482
COMM MOVJ C00384 BC00384 VJ=100.00  +MOVJ EC00384 VJ=100.00
COMM MOVJ C00385 BC00385 VJ=100.00  +MOVJ EC00385 VJ=100.00
COMM '10
COMM '11
COMM 'Path W3484
COMM SFTOF3D
COMM SFTON3D P025
COMM MOVJ C00386 BC00386 VJ=100.00  +MOVJ EC00386 VJ=100.00
COMM SMOVL C00387 BC00387 V=800.0  +MOVJ EC00387
COMM SMOVL C00388 BC00388 V=150.0 PL=0  +MOVJ EC00388
COMM ARCON
COMM SMOVL C00389 BC00389 V=10.0  +MOVJ EC00389
COMM SMOVL C00390 BC00390 V=10.0  +MOVJ EC00390
COMM ARCOF
COMM SMOVL C00391 BC00391 V=800.0  +MOVJ EC00391
COMM SMOVL C00392 BC00392 V=1000.0  +MOVJ EC00392
COMM SFTOF3D
COMM 'EndPath W3484
COMM MOVJ C00393 BC00393 VJ=100.00  +MOVJ EC00393 VJ=100.00
COMM 'brak dostepu offset drutu 1cm
COMM 'Path W3483
COMM SFTOF3D
COMM SFTON3D P025
COMM MOVJ C00394 BC00394 VJ=100.00  +MOVJ EC00394 VJ=100.00
COMM SMOVL C00395 BC00395 V=800.0  +MOVJ EC00395
COMM SMOVL C00396 BC00396 V=166.7 PL=0  +MOVJ EC00396
COMM ARCON
COMM SMOVL C00397 BC00397 V=10.0  +MOVJ EC00397
COMM ARCOF
COMM SMOVL C00398 BC00398 V=800.0  +MOVJ EC00398
COMM SMOVL C00399 BC00399 V=1000.0  +MOVJ EC00399
COMM SFTOF3D
COMM 'EndPath W3483
COMM MOVJ C00400 BC00400 VJ=100.00  +MOVJ EC00400 VJ=100.00
COMM MOVJ C00401 BC00401 VJ=100.00  +MOVJ EC00401 VJ=100.00
COMM MOVJ C00402 BC00402 VJ=100.00  +MOVJ EC00402 VJ=100.00
COMM 'Path W4854
COMM SFTOF3D
COMM SFTON3D P073
COMM MOVJ C00403 BC00403 VJ=100.00  +MOVJ EC00403 VJ=100.00
COMM SMOVL C00404 BC00404 V=800.0  +MOVJ EC00404
COMM SMOVL C00405 BC00405 V=150.0 PL=0  +MOVJ EC00405
COMM MACRO1 MJ#(0) ARGF9
COMM ARCON
COMM SMOVL C00406 BC00406 V=9.2  +MOVJ EC00406
COMM SFTON3D P074
COMM SMOVL C00407 BC00407 V=9.2  +MOVJ EC00407
COMM SMOVL C00408 BC00408 V=9.2  +MOVJ EC00408
COMM ARCOF
COMM SMOVL C00409 BC00409 V=800.0  +MOVJ EC00409
COMM SMOVL C00410 BC00410 V=1000.0  +MOVJ EC00410
COMM SFTOF3D
COMM 'EndPath W4854
COMM '12
COMM MOVJ C00411 BC00411 VJ=100.00  +MOVJ EC00411 VJ=100.00
COMM MOVJ C00412 BC00412 VJ=100.00  +MOVJ EC00412 VJ=100.00
COMM MOVJ C00413 BC00413 VJ=100.00  +MOVJ EC00413 VJ=100.00
COMM 'Path W3485
COMM SFTOF3D
COMM SFTON3D P034
COMM MOVJ C00414 BC00414 VJ=100.00  +MOVJ EC00414 VJ=100.00
COMM SMOVL C00415 BC00415 V=800.0  +MOVJ EC00415
COMM SMOVL C00416 BC00416 V=150.0 PL=0  +MOVJ EC00416
COMM MACRO1 MJ#(0) ARGF14
COMM ARCON
COMM SMOVL C00417 BC00417 V=10.0  +MOVJ EC00417
COMM SMOVL C00418 BC00418 V=10.0  +MOVJ EC00418
COMM SMOVL C00419 BC00419 V=10.0  +MOVJ EC00419
COMM ARCOF
COMM SMOVL C00420 BC00420 V=800.0  +MOVJ EC00420
COMM SMOVL C00421 BC00421 V=1000.0  +MOVJ EC00421
COMM SFTOF3D
COMM MOVJ C00422 BC00422 VJ=80.00  +MOVJ EC00422 VJ=80.00
COMM MOVJ C00423 BC00423 VJ=80.00  +MOVJ EC00423 VJ=80.00
COMM MOVJ C00424 BC00424 VJ=80.00  +MOVJ EC00424 VJ=80.00
COMM MACRO1 MJ#(0) ARGF6
COMM SFTON3D P063
COMM SMOVL C00425 BC00425 V=166.7  +MOVJ EC00425
COMM ARCON
